KUKA KRL program: EPS_2_25694_BP04_A_20251117072358.src

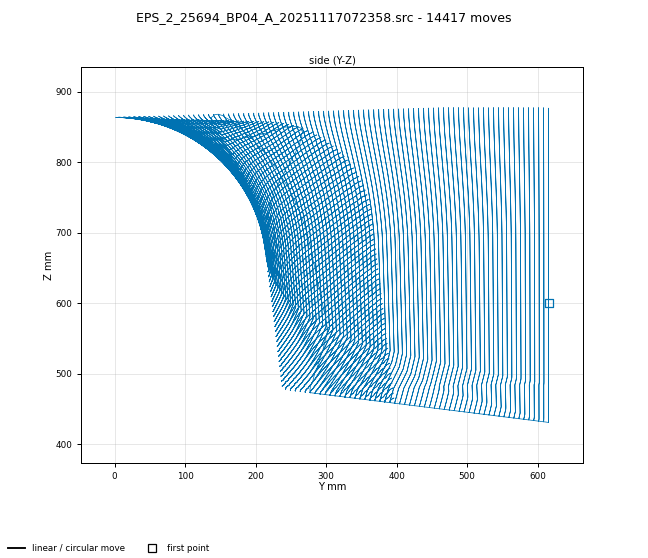
[picture p0: tool path of EPS_2_25694_BP04_A_20251117072358.src, 14417 of 14419 moves have a stored position in this frame; points joined in program order, loops and branches not executed]
&ACCESS RVP
&REL 4
&COMMENT QRS 19112012
&PARAM EDITMASK = *
DEF PART()
EXT BAS (BAS_COMMAND :IN,REAL :IN )
INT I
BAS (#INITMOV,0 )

;KUKA QRS Post kuka4.cps  Date:22-06-2017 !

File_ID=2911

QRS_PRE_INIT()

;Init var - Until changes are made in qrs_pre_init
Outlet_Square_prg=0
Inlet_1_Square_prg=0
Inlet_2_Square_prg=0
Inlet_3_Square_prg=0
Inlet_4_Square_prg=0
Inlet_5_Square_prg=0

Outlet_1={X 0.000, Y 466.000, Z 687.000, B 0.000, E1 0.000 }
Inlet_1={X 0.000, Y 508.730, Z 662.000, B 0.000, E1 180.000 }
Outlet_1_type=381
Inlet_1_type=0
;QRS#1=Sidecore dimensions
;QRS#2=375-15" Concrete
;QRS#3=DeadEnd 381
;QRS#4=
;QRS#5=
;QRS#6=
;QRS#7=
;QRS#8=
;QRS#9=24L PSX-2
;QRS#10=

;QRS#11=
;QRS#12=
;QRS#13=
;QRS#14=
;QRS#15=
;QRS#16=1220x127x1219 4'
;QRS#17=EPS Height
;QRS#18=877,5
;QRS#19=*
;QRS#20= UPDATED VERSION 22-06-2017
;QRS#21=*
Outlet_Square=0150
Inlet_1_Square=00
Inlet_2_Square=0
Inlet_3_Square=0
Inlet_4_Square=0
Inlet_5_Square=0
Mill_Square=1
Outlet_Square_Prg=261
Inlet_1_Square_prg=0

QRS_INIT()

$ADVANCE=5

; T1
PTP {E1 173.596,E2 173.596}
PTP {X 0,Y 615.505,A -85,B 0,C 180,E1 173.596,E2 173.596,E3 0,E4 0,E5 0,E6 0}
QRS_SPEED_INIT()
LIN {X 0,Y 615.505,Z 600,A -85,B 0,C 180,E1 173.596,E2 173.596,E3 0,E4 0,E5 0,E6 0} C_VEL
LIN {X 0,Y 615.505,Z 441.122,A -85,B 0,C 180,E1 173.596,E2 173.596} C_VEL
LIN {X 0,Y 615.505,Z 432.953,A -85,B 0,C 180,E1 173.596,E2 173.596} C_VEL
LIN {X 0,Y 615.487,Z 430.953,A -85,B 0,C 180,E1 173.41,E2 173.41} C_VEL
LIN {X 0,Y 615.475,Z 430.938,A -85,B 0,C 180,E1 170.801,E2 170.801} C_VEL
LIN {X 0,Y 615.486,Z 430.932,A -85,B 0,C 180,E1 168.139,E2 168.139} C_VEL
LIN {X 0,Y 615.48,Z 430.947,A -85,B 0,C 180,E1 165.451,E2 165.451} C_VEL
LIN {X 0,Y 615.476,Z 430.939,A -85,B 0,C 180,E1 162.729,E2 162.729} C_VEL
LIN {X 0,Y 615.485,Z 430.933,A -85,B 0,C 180,E1 159.967,E2 159.967} C_VEL
LIN {X 0,Y 615.486,Z 430.952,A -85,B 0,C 180,E1 157.156,E2 157.156} C_VEL
LIN {X 0,Y 615.484,Z 430.933,A -85,B 0,C 180,E1 154.284,E2 154.284} C_VEL
LIN {X 0,Y 615.476,Z 430.939,A -85,B 0,C 180,E1 151.549,E2 151.549} C_VEL
LIN {X 0,Y 615.483,Z 430.951,A -85,B 0,C 180,E1 148.912,E2 148.912} C_VEL
LIN {X 0,Y 615.496,Z 430.929,A -85,B 0,C 180,E1 145.979,E2 145.979} C_VEL
LIN {X 0,Y 615.487,Z 430.946,A -85,B 0,C 180,E1 143.062,E2 143.062} C_VEL
LIN {X 0,Y 615.474,Z 430.938,A -85,B 0,C 180,E1 140.249,E2 140.249} C_VEL
LIN {X 0,Y 615.488,Z 430.931,A -85,B 0,C 180,E1 137.648,E2 137.648} C_VEL
LIN {X 0,Y 615.48,Z 430.948,A -85,B 0,C 180,E1 134.931,E2 134.931} C_VEL
LIN {X 0,Y 615.477,Z 430.936,A -85,B 0,C 180,E1 132.08,E2 132.08} C_VEL
LIN {X 0,Y 615.493,Z 430.93,A -85,B 0,C 180,E1 129.749,E2 129.749} C_VEL
LIN {X 0,Y 615.478,Z 430.944,A -85,B 0,C 180,E1 126.936,E2 126.936} C_VEL
LIN {X 0,Y 615.49,Z 430.948,A -85,B 0,C 180,E1 124.702,E2 124.702} C_VEL
LIN {X 0,Y 615.484,Z 430.946,A -85,B 0,C 180,E1 122.331,E2 122.331} C_VEL
LIN {X 0,Y 615.493,Z 430.93,A -85,B 0,C 180,E1 119.405,E2 119.405} C_VEL
LIN {X 0,Y 615.491,Z 430.952,A -85,B 0,C 180,E1 116.443,E2 116.443} C_VEL
LIN {X 0,Y 615.487,Z 430.932,A -85,B 0,C 180,E1 113.556,E2 113.556} C_VEL
LIN {X 0,Y 615.477,Z 430.942,A -85,B 0,C 180,E1 110.731,E2 110.731} C_VEL
LIN {X 0,Y 615.478,Z 430.943,A -85,B 0,C 180,E1 107.957,E2 107.957} C_VEL
LIN {X 0,Y 615.488,Z 430.931,A -85,B 0,C 180,E1 105.226,E2 105.226} C_VEL
LIN {X 0,Y 615.479,Z 430.943,A -85,B 0,C 180,E1 102.53,E2 102.53} C_VEL
LIN {X 0,Y 615.48,Z 430.943,A -85,B 0,C 180,E1 99.862,E2 99.862} C_VEL
LIN {X 0,Y 615.489,Z 430.931,A -85,B 0,C 180,E1 97.215,E2 97.215} C_VEL
LIN {X 0,Y 615.476,Z 430.939,A -85,B 0,C 180,E1 94.585,E2 94.585} C_VEL
LIN {X 0,Y 615.493,Z 430.949,A -85,B 0,C 180,E1 91.963,E2 91.963} C_VEL
LIN {X 0,Y 615.474,Z 430.937,A -85,B 0,C 180,E1 89.346,E2 89.346} C_VEL
LIN {X 0,Y 615.484,Z 430.933,A -85,B 0,C 180,E1 86.727,E2 86.727} C_VEL
LIN {X 0,Y 615.484,Z 430.946,A -85,B 0,C 180,E1 84.102,E2 84.102} C_VEL
LIN {X 0,Y 615.477,Z 430.941,A -85,B 0,C 180,E1 81.463,E2 81.463} C_VEL
LIN {X 0,Y 615.497,Z 430.929,A -85,B 0,C 180,E1 78.807,E2 78.807} C_VEL
LIN {X 0,Y 615.48,Z 430.944,A -85,B 0,C 180,E1 76.068,E2 76.068} C_VEL
LIN {X 0,Y 615.477,Z 430.944,A -85,B 0,C 180,E1 73.413,E2 73.413} C_VEL
LIN {X 0,Y 615.485,Z 430.931,A -85,B 0,C 180,E1 70.662,E2 70.662} C_VEL
LIN {X 0,Y 615.478,Z 430.946,A -85,B 0,C 180,E1 67.864,E2 67.864} C_VEL
LIN {X 0,Y 615.475,Z 430.938,A -85,B 0,C 180,E1 65.008,E2 65.008} C_VEL
LIN {X 0,Y 615.481,Z 430.934,A -85,B 0,C 180,E1 62.823,E2 62.823} C_VEL
LIN {X 0,Y 615.476,Z 430.936,A -85,B 0,C 180,E1 60.206,E2 60.206} C_VEL
LIN {X 0,Y 615.489,Z 430.949,A -85,B 0,C 180,E1 57.543,E2 57.543} C_VEL
LIN {X 0,Y 615.483,Z 430.945,A -85,B 0,C 180,E1 55.186,E2 55.186} C_VEL
LIN {X 0,Y 615.474,Z 430.937,A -85,B 0,C 180,E1 52.758,E2 52.758} C_VEL
LIN {X 0,Y 615.476,Z 430.937,A -85,B 0,C 180,E1 49.912,E2 49.912} C_VEL
LIN {X 0,Y 615.478,Z 430.942,A -85,B 0,C 180,E1 47.647,E2 47.647} C_VEL
LIN {X 0,Y 615.48,Z 430.943,A -85,B 0,C 180,E1 44.932,E2 44.932} C_VEL
LIN {X 0,Y 615.49,Z 430.931,A -85,B 0,C 180,E1 42.082,E2 42.082} C_VEL
LIN {X 0,Y 615.493,Z 430.948,A -85,B 0,C 180,E1 39.064,E2 39.064} C_VEL
LIN {X 0,Y 615.479,Z 430.935,A -85,B 0,C 180,E1 36.425,E2 36.425} C_VEL
LIN {X 0,Y 615.476,Z 430.94,A -85,B 0,C 180,E1 33.535,E2 33.535} C_VEL
LIN {X 0,Y 615.485,Z 430.95,A -85,B 0,C 180,E1 30.919,E2 30.919} C_VEL
LIN {X 0,Y 615.476,Z 430.939,A -85,B 0,C 180,E1 28.451,E2 28.451} C_VEL
LIN {X 0,Y 615.484,Z 430.933,A -85,B 0,C 180,E1 25.716,E2 25.716} C_VEL
LIN {X 0,Y 615.486,Z 430.952,A -85,B 0,C 180,E1 22.844,E2 22.844} C_VEL
LIN {X 0,Y 615.485,Z 430.933,A -85,B 0,C 180,E1 20.033,E2 20.033} C_VEL
LIN {X 0,Y 615.476,Z 430.939,A -85,B 0,C 180,E1 17.271,E2 17.271} C_VEL
LIN {X 0,Y 615.484,Z 430.947,A -85,B 0,C 180,E1 14.549,E2 14.549} C_VEL
LIN {X 0,Y 615.486,Z 430.932,A -85,B 0,C 180,E1 11.861,E2 11.861} C_VEL
LIN {X 0,Y 615.475,Z 430.938,A -85,B 0,C 180,E1 9.199,E2 9.199} C_VEL
LIN {X 0,Y 615.489,Z 430.951,A -85,B 0,C 180,E1 6.556,E2 6.556} C_VEL
LIN {X 0,Y 615.477,Z 430.936,A -85,B 0,C 180,E1 3.928,E2 3.928} C_VEL
LIN {X 0,Y 615.484,Z 430.933,A -85,B 0,C 180,E1 1.308,E2 1.308} C_VEL
LIN {X 0,Y 615.483,Z 430.945,A -85,B 0,C 180,E1 -1.309,E2 -1.309} C_VEL
LIN {X 0,Y 615.478,Z 430.942,A -85,B 0,C 180,E1 -3.929,E2 -3.929} C_VEL
LIN {X 0,Y 615.487,Z 430.931,A -85,B 0,C 180,E1 -6.589,E2 -6.589} C_VEL
LIN {X 0,Y 615.474,Z 430.94,A -85,B 0,C 180,E1 -9.199,E2 -9.199} C_VEL
LIN {X 0,Y 615.484,Z 430.948,A -85,B 0,C 180,E1 -11.861,E2 -11.861} C_VEL
LIN {X 0,Y 615.48,Z 430.934,A -85,B 0,C 180,E1 -14.549,E2 -14.549} C_VEL
LIN {X 0,Y 615.475,Z 430.939,A -85,B 0,C 180,E1 -17.271,E2 -17.271} C_VEL
LIN {X 0,Y 615.484,Z 430.946,A -85,B 0,C 180,E1 -20.033,E2 -20.033} C_VEL
LIN {X 0,Y 615.486,Z 430.931,A -85,B 0,C 180,E1 -22.845,E2 -22.845} C_VEL
LIN {X 0,Y 615.483,Z 430.945,A -85,B 0,C 180,E1 -25.716,E2 -25.716} C_VEL
LIN {X 0,Y 615.477,Z 430.94,A -85,B 0,C 180,E1 -28.451,E2 -28.451} C_VEL
LIN {X 0,Y 615.483,Z 430.932,A -85,B 0,C 180,E1 -31.088,E2 -31.088} C_VEL
LIN {X 0,Y 615.495,Z 430.949,A -85,B 0,C 180,E1 -34.021,E2 -34.021} C_VEL
LIN {X 0,Y 615.486,Z 430.932,A -85,B 0,C 180,E1 -36.938,E2 -36.938} C_VEL
LIN {X 0,Y 615.476,Z 430.941,A -85,B 0,C 180,E1 -39.751,E2 -39.751} C_VEL
LIN {X 0,Y 615.489,Z 430.947,A -85,B 0,C 180,E1 -42.353,E2 -42.353} C_VEL
LIN {X 0,Y 615.48,Z 430.934,A -85,B 0,C 180,E1 -45.069,E2 -45.069} C_VEL
LIN {X 0,Y 615.476,Z 430.942,A -85,B 0,C 180,E1 -47.921,E2 -47.921} C_VEL
LIN {X 0,Y 615.491,Z 430.948,A -85,B 0,C 180,E1 -50.251,E2 -50.251} C_VEL
LIN {X 0,Y 615.48,Z 430.935,A -85,B 0,C 180,E1 -53.064,E2 -53.064} C_VEL
LIN {X 0,Y 615.49,Z 430.931,A -85,B 0,C 180,E1 -55.299,E2 -55.299} C_VEL
LIN {X 0,Y 615.484,Z 430.933,A -85,B 0,C 180,E1 -57.669,E2 -57.669} C_VEL
LIN {X 0,Y 615.498,Z 431.074,A -85,B 0,C 180,E1 -60.595,E2 -60.595} C_VEL
LIN {X 0,Y 615.496,Z 431.86,A -85,B 0,C 180,E1 -60.782,E2 -60.782} C_VEL
LIN {X 0,Y 615.493,Z 454.299,A -85,B 0,C 180,E1 -63.557,E2 -63.557} C_VEL
LIN {X 0,Y 615.477,Z 476.35,A -85,B 0,C 180,E1 -66.219,E2 -66.219} C_VEL
LIN {X 0,Y 615.491,Z 484.19,A -85,B 0,C 180,E1 -67.134,E2 -67.134} C_VEL
LIN {X 0,Y 615.489,Z 494.25,A -85,B 0,C 180,E1 -67.28,E2 -67.28} C_VEL
LIN {X 0,Y 615.488,Z 696.741,A -85,B 0,C 180,E1 -69.786,E2 -69.786} C_VEL
LIN {X 0,Y 615.493,Z 712.21,A -85,B 0,C 180,E1 -70.098,E2 -70.098} C_VEL
LIN {X 0,Y 615.492,Z 727.984,A -85,B 0,C 180,E1 -70.533,E2 -70.533} C_VEL
LIN {X 0,Y 615.492,Z 743.625,A -85,B 0,C 180,E1 -71.095,E2 -71.095} C_VEL
LIN {X 0,Y 615.497,Z 759.271,A -85,B 0,C 180,E1 -71.8,E2 -71.8} C_VEL
LIN {X 0,Y 615.499,Z 774.742,A -85,B 0,C 180,E1 -72.645,E2 -72.645} C_VEL
LIN {X 0,Y 615.497,Z 788.923,A -85,B 0,C 180,E1 -73.565,E2 -73.565} C_VEL
LIN {X 0,Y 615.497,Z 802.468,A -85,B 0,C 180,E1 -74.605,E2 -74.605} C_VEL
LIN {X 0,Y 615.496,Z 815.245,A -85,B 0,C 180,E1 -75.759,E2 -75.759} C_VEL
LIN {X 0,Y 615.491,Z 826.671,A -85,B 0,C 180,E1 -76.967,E2 -76.967} C_VEL
LIN {X 0,Y 615.489,Z 837.477,A -85,B 0,C 180,E1 -78.307,E2 -78.307} C_VEL
LIN {X 0,Y 615.49,Z 846.606,A -85,B 0,C 180,E1 -79.64,E2 -79.64} C_VEL
LIN {X 0,Y 615.49,Z 855.145,A -85,B 0,C 180,E1 -81.133,E2 -81.133} C_VEL
LIN {X 0,Y 615.492,Z 862.719,A -85,B 0,C 180,E1 -82.785,E2 -82.785} C_VEL
LIN {X 0,Y 615.487,Z 867.467,A -85,B 0,C 180,E1 -84.102,E2 -84.102} C_VEL
LIN {X 0,Y 615.489,Z 871.26,A -85,B 0,C 180,E1 -85.416,E2 -85.416} C_VEL
LIN {X 0,Y 615.493,Z 873.996,A -85,B 0,C 180,E1 -86.727,E2 -86.727} C_VEL
LIN {X 0,Y 615.494,Z 875.835,A -85,B 0,C 180,E1 -88.037,E2 -88.037} C_VEL
LIN {X 0,Y 615.491,Z 876.738,A -85,B 0,C 180,E1 -89.346,E2 -89.346} C_VEL
LIN {X 0,Y 615.491,Z 876.738,A -85,B 0,C 180,E1 -90.654,E2 -90.654} C_VEL
LIN {X 0,Y 615.494,Z 875.835,A -85,B 0,C 180,E1 -91.963,E2 -91.963} C_VEL
LIN {X 0,Y 615.493,Z 873.996,A -85,B 0,C 180,E1 -93.273,E2 -93.273} C_VEL
LIN {X 0,Y 615.489,Z 871.26,A -85,B 0,C 180,E1 -94.584,E2 -94.584} C_VEL
LIN {X 0,Y 615.491,Z 866.415,A -85,B 0,C 180,E1 -96.227,E2 -96.227} C_VEL
LIN {X 0,Y 615.486,Z 861.303,A -85,B 0,C 180,E1 -97.545,E2 -97.545} C_VEL
LIN {X 0,Y 615.49,Z 855.145,A -85,B 0,C 180,E1 -98.867,E2 -98.867} C_VEL
LIN {X 0,Y 615.489,Z 845.582,A -85,B 0,C 180,E1 -100.527,E2 -100.527} C_VEL
LIN {X 0,Y 615.492,Z 836.244,A -85,B 0,C 180,E1 -101.86,E2 -101.86} C_VEL
LIN {X 0,Y 615.491,Z 826.671,A -85,B 0,C 180,E1 -103.033,E2 -103.033} C_VEL
LIN {X 0,Y 615.496,Z 815.245,A -85,B 0,C 180,E1 -104.241,E2 -104.241} C_VEL
LIN {X 0,Y 615.497,Z 802.468,A -85,B 0,C 180,E1 -105.395,E2 -105.395} C_VEL
LIN {X 0,Y 615.495,Z 788.932,A -85,B 0,C 180,E1 -106.434,E2 -106.434} C_VEL
LIN {X 0,Y 615.498,Z 774.742,A -85,B 0,C 180,E1 -107.355,E2 -107.355} C_VEL
LIN {X 0,Y 615.497,Z 759.271,A -85,B 0,C 180,E1 -108.2,E2 -108.2} C_VEL
LIN {X 0,Y 615.492,Z 743.625,A -85,B 0,C 180,E1 -108.905,E2 -108.905} C_VEL
LIN {X 0,Y 615.492,Z 727.984,A -85,B 0,C 180,E1 -109.467,E2 -109.467} C_VEL
LIN {X 0,Y 615.493,Z 712.21,A -85,B 0,C 180,E1 -109.902,E2 -109.902} C_VEL
LIN {X 0,Y 615.489,Z 695.6,A -85,B 0,C 180,E1 -110.23,E2 -110.23} C_VEL
LIN {X 0,Y 615.49,Z 484.677,A -85,B 0,C 180,E1 -112.844,E2 -112.844} C_VEL
LIN {X 0,Y 615.493,Z 483.482,A -85,B 0,C 180,E1 -112.933,E2 -112.933} C_VEL
LIN {X 0,Y 615.482,Z 460.283,A -85,B 0,C 180,E1 -115.715,E2 -115.715} C_VEL
LIN {X 0,Y 615.495,Z 436.348,A -85,B 0,C 180,E1 -118.657,E2 -118.657} C_VEL
LIN {X 0,Y 615.496,Z 431.31,A -85,B 0,C 180,E1 -119.311,E2 -119.311} C_VEL
LIN {X 0,Y 615.477,Z 430.936,A -85,B 0,C 180,E1 -120.16,E2 -120.16} C_VEL
LIN {X 0,Y 615.489,Z 430.931,A -85,B 0,C 180,E1 -122.457,E2 -122.457} C_VEL
LIN {X 0,Y 615.483,Z 430.933,A -85,B 0,C 180,E1 -124.814,E2 -124.814} C_VEL
LIN {X 0,Y 615.477,Z 430.942,A -85,B 0,C 180,E1 -127.242,E2 -127.242} C_VEL
LIN {X 0,Y 615.476,Z 430.941,A -85,B 0,C 180,E1 -130.088,E2 -130.088} C_VEL
LIN {X 0,Y 615.477,Z 430.936,A -85,B 0,C 180,E1 -132.353,E2 -132.353} C_VEL
LIN {X 0,Y 615.48,Z 430.935,A -85,B 0,C 180,E1 -135.068,E2 -135.068} C_VEL
LIN {X 0,Y 615.489,Z 430.947,A -85,B 0,C 180,E1 -137.918,E2 -137.918} C_VEL
LIN {X 0,Y 615.476,Z 430.941,A -85,B 0,C 180,E1 -140.249,E2 -140.249} C_VEL
LIN {X 0,Y 615.486,Z 430.932,A -85,B 0,C 180,E1 -143.062,E2 -143.062} C_VEL
LIN {X 0,Y 615.495,Z 430.949,A -85,B 0,C 180,E1 -145.979,E2 -145.979} C_VEL
LIN {X 0,Y 615.481,Z 430.933,A -85,B 0,C 180,E1 -148.913,E2 -148.913} C_VEL
LIN {X 0,Y 615.477,Z 430.94,A -85,B 0,C 180,E1 -151.549,E2 -151.549} C_VEL
LIN {X 0,Y 615.483,Z 430.945,A -85,B 0,C 180,E1 -154.284,E2 -154.284} C_VEL
LIN {X 0,Y 615.486,Z 430.931,A -85,B 0,C 180,E1 -157.155,E2 -157.155} C_VEL
LIN {X 0,Y 615.484,Z 430.946,A -85,B 0,C 180,E1 -159.967,E2 -159.967} C_VEL
LIN {X 0,Y 615.475,Z 430.939,A -85,B 0,C 180,E1 -162.729,E2 -162.729} C_VEL
LIN {X 0,Y 615.48,Z 430.934,A -85,B 0,C 180,E1 -165.451,E2 -165.451} C_VEL
LIN {X 0,Y 615.484,Z 430.948,A -85,B 0,C 180,E1 -168.139,E2 -168.139} C_VEL
LIN {X 0,Y 615.474,Z 430.94,A -85,B 0,C 180,E1 -170.801,E2 -170.801} C_VEL
LIN {X 0,Y 615.488,Z 430.931,A -85,B 0,C 180,E1 -173.443,E2 -173.443} C_VEL
LIN {X 0,Y 615.478,Z 430.942,A -85,B 0,C 180,E1 -176.071,E2 -176.071} C_VEL
LIN {X 0,Y 615.483,Z 430.945,A -85,B 0,C 180,E1 -178.691,E2 -178.691} C_VEL
LIN {X 0,Y 615.484,Z 430.933,A -85,B 0,C 180,E1 -181.308,E2 -181.308} C_VEL
LIN {X 0,Y 615.477,Z 430.936,A -85,B 0,C 180,E1 -183.928,E2 -183.928} C_VEL
LIN {X 0,Y 615.487,Z 430.953,A -85,B 0,C 180,E1 -186.59,E2 -186.59} C_VEL
LIN {X 0,Y 614.804,Z 431.086,A -85,B 0,C 180,E1 -187.135,E2 -187.135} C_VEL
LIN {X 0,Y 611.961,Z 431.501,A -85,B 0,C 180,E1 -188.021,E2 -188.021} C_VEL
LIN {X 0,Y 609.57,Z 431.811,A -85,B 0,C 180,E1 -188.734,E2 -188.734} C_VEL
LIN {X 0,Y 608.538,Z 431.928,A -85,B 0,C 180,E1 -189.284,E2 -189.284} C_VEL
LIN {X 0,Y 608.451,Z 431.937,A -85,B 0,C 180,E1 -189.47,E2 -189.47} C_VEL
LIN {X 0,Y 608.46,Z 431.937,A -85,B 0,C 180,E1 -192,E2 -192} C_VEL
LIN {X 0,Y 608.467,Z 431.946,A -85,B 0,C 180,E1 -194.72,E2 -194.72} C_VEL
LIN {X 0,Y 608.445,Z 431.939,A -85,B 0,C 180,E1 -197.477,E2 -197.477} C_VEL
LIN {X 0,Y 608.459,Z 431.938,A -85,B 0,C 180,E1 -200.274,E2 -200.274} C_VEL
LIN {X 0,Y 608.447,Z 431.944,A -85,B 0,C 180,E1 -203.124,E2 -203.124} C_VEL
LIN {X 0,Y 608.465,Z 431.935,A -85,B 0,C 180,E1 -205.722,E2 -205.722} C_VEL
LIN {X 0,Y 608.445,Z 431.938,A -85,B 0,C 180,E1 -208.267,E2 -208.267} C_VEL
LIN {X 0,Y 608.47,Z 431.938,A -85,B 0,C 180,E1 -210.544,E2 -210.544} C_VEL
LIN {X 0,Y 608.45,Z 431.945,A -85,B 0,C 180,E1 -212.88,E2 -212.88} C_VEL
LIN {X 0,Y 608.434,Z 431.947,A -85,B 0,C 180,E1 -215.278,E2 -215.278} C_VEL
LIN {X 0,Y 608.47,Z 431.936,A -85,B 0,C 180,E1 -217.746,E2 -217.746} C_VEL
LIN {X 0,Y 608.473,Z 431.934,A -85,B 0,C 180,E1 -220.333,E2 -220.333} C_VEL
LIN {X 0,Y 608.483,Z 431.943,A -85,B 0,C 180,E1 -223.311,E2 -223.311} C_VEL
LIN {X 0,Y 608.465,Z 431.935,A -85,B 0,C 180,E1 -226.131,E2 -226.131} C_VEL
LIN {X 0,Y 608.447,Z 431.94,A -85,B 0,C 180,E1 -228.824,E2 -228.824} C_VEL
LIN {X 0,Y 608.462,Z 431.946,A -85,B 0,C 180,E1 -231.413,E2 -231.413} C_VEL
LIN {X 0,Y 608.471,Z 431.937,A -85,B 0,C 180,E1 -233.951,E2 -233.951} C_VEL
LIN {X 0,Y 608.466,Z 431.935,A -85,B 0,C 180,E1 -236.33,E2 -236.33} C_VEL
LIN {X 0,Y 608.471,Z 431.935,A -85,B 0,C 180,E1 -238.728,E2 -238.728} C_VEL
LIN {X 0,Y 608.472,Z 431.943,A -85,B 0,C 180,E1 -241.379,E2 -241.379} C_VEL
LIN {X 0,Y 608.467,Z 431.936,A -85,B 0,C 180,E1 -244.279,E2 -244.279} C_VEL
LIN {X 0,Y 608.445,Z 431.938,A -85,B 0,C 180,E1 -246.876,E2 -246.876} C_VEL
LIN {X 0,Y 608.463,Z 431.941,A -85,B 0,C 180,E1 -249.321,E2 -249.321} C_VEL
LIN {X 0,Y 608.442,Z 431.947,A -85,B 0,C 180,E1 -251.828,E2 -251.828} C_VEL
LIN {X 0,Y 608.47,Z 431.935,A -85,B 0,C 180,E1 -254.594,E2 -254.594} C_VEL
LIN {X 0,Y 608.472,Z 431.938,A -85,B 0,C 180,E1 -257.323,E2 -257.323} C_VEL
LIN {X 0,Y 608.449,Z 431.945,A -85,B 0,C 180,E1 -260.023,E2 -260.023} C_VEL
LIN {X 0,Y 608.483,Z 431.933,A -85,B 0,C 180,E1 -262.701,E2 -262.701} C_VEL
LIN {X 0,Y 608.446,Z 431.94,A -85,B 0,C 180,E1 -265.362,E2 -265.362} C_VEL
LIN {X 0,Y 608.463,Z 431.946,A -85,B 0,C 180,E1 -268.014,E2 -268.014} C_VEL
LIN {X 0,Y 608.469,Z 431.936,A -85,B 0,C 180,E1 -270.662,E2 -270.662} C_VEL
LIN {X 0,Y 608.477,Z 431.934,A -85,B 0,C 180,E1 -273.311,E2 -273.311} C_VEL
LIN {X 0,Y 608.457,Z 431.945,A -85,B 0,C 180,E1 -275.967,E2 -275.967} C_VEL
LIN {X 0,Y 608.45,Z 431.94,A -85,B 0,C 180,E1 -278.636,E2 -278.636} C_VEL
LIN {X 0,Y 608.48,Z 431.933,A -85,B 0,C 180,E1 -281.323,E2 -281.323} C_VEL
LIN {X 0,Y 608.464,Z 431.943,A -85,B 0,C 180,E1 -284.037,E2 -284.037} C_VEL
LIN {X 0,Y 608.472,Z 431.937,A -85,B 0,C 180,E1 -286.783,E2 -286.783} C_VEL
LIN {X 0,Y 608.449,Z 431.938,A -85,B 0,C 180,E1 -289.57,E2 -289.57} C_VEL
LIN {X 0,Y 608.454,Z 431.946,A -85,B 0,C 180,E1 -292.476,E2 -292.476} C_VEL
LIN {X 0,Y 608.45,Z 431.945,A -85,B 0,C 180,E1 -294.571,E2 -294.571} C_VEL
LIN {X 0,Y 608.473,Z 431.935,A -85,B 0,C 180,E1 -297.207,E2 -297.207} C_VEL
LIN {X 0,Y 608.457,Z 431.939,A -85,B 0,C 180,E1 -299.971,E2 -299.971} C_VEL
LIN {X 0,Y 608.462,Z 431.947,A -85,B 0,C 180,E1 -302.523,E2 -302.523} C_VEL
LIN {X 0,Y 608.448,Z 431.938,A -85,B 0,C 180,E1 -305.276,E2 -305.276} C_VEL
LIN {X 0,Y 608.46,Z 431.936,A -85,B 0,C 180,E1 -307.746,E2 -307.746} C_VEL
LIN {X 0,Y 608.445,Z 431.943,A -85,B 0,C 180,E1 -310.329,E2 -310.329} C_VEL
LIN {X 0,Y 608.446,Z 431.944,A -85,B 0,C 180,E1 -312.959,E2 -312.959} C_VEL
LIN {X 0,Y 608.459,Z 431.936,A -85,B 0,C 180,E1 -315.735,E2 -315.735} C_VEL
LIN {X 0,Y 608.456,Z 431.945,A -85,B 0,C 180,E1 -318.657,E2 -318.657} C_VEL
LIN {X 0,Y 608.466,Z 431.937,A -85,B 0,C 180,E1 -321.412,E2 -321.412} C_VEL
LIN {X 0,Y 608.469,Z 431.935,A -85,B 0,C 180,E1 -323.95,E2 -323.95} C_VEL
LIN {X 0,Y 608.459,Z 431.937,A -85,B 0,C 180,E1 -326.329,E2 -326.329} C_VEL
LIN {X 0,Y 608.468,Z 431.941,A -85,B 0,C 180,E1 -328.727,E2 -328.727} C_VEL
LIN {X 0,Y 608.465,Z 431.94,A -85,B 0,C 180,E1 -331.379,E2 -331.379} C_VEL
LIN {X 0,Y 608.44,Z 431.938,A -85,B 0,C 180,E1 -333.965,E2 -333.965} C_VEL
LIN {X 0,Y 608.464,Z 431.935,A -85,B 0,C 180,E1 -336.155,E2 -336.155} C_VEL
LIN {X 0,Y 608.453,Z 431.945,A -85,B 0,C 180,E1 -339.019,E2 -339.019} C_VEL
LIN {X 0,Y 608.449,Z 431.939,A -85,B 0,C 180,E1 -341.828,E2 -341.828} C_VEL
LIN {X 0,Y 608.462,Z 431.936,A -85,B 0,C 180,E1 -344.594,E2 -344.594} C_VEL
LIN {X 0,Y 608.472,Z 431.945,A -85,B 0,C 180,E1 -347.323,E2 -347.323} C_VEL
LIN {X 0,Y 608.454,Z 431.938,A -85,B 0,C 180,E1 -350.023,E2 -350.023} C_VEL
LIN {X 0,Y 608.455,Z 431.937,A -85,B 0,C 180,E1 -352.701,E2 -352.701} C_VEL
LIN {X 0,Y 608.465,Z 431.945,A -85,B 0,C 180,E1 -355.363,E2 -355.363} C_VEL
LIN {X 0,Y 608.446,Z 431.94,A -85,B 0,C 180,E1 -358.014,E2 -358.014} C_VEL
LIN {X 0,Y 608.478,Z 431.934,A -85,B 0,C 180,E1 -360.662,E2 -360.662} C_VEL
LIN {X 0,Y 608.472,Z 431.941,A -85,B 0,C 180,E1 -363.311,E2 -363.311} C_VEL
LIN {X 0,Y 608.453,Z 431.941,A -85,B 0,C 180,E1 -365.967,E2 -365.967} C_VEL
LIN {X 0,Y 608.457,Z 431.936,A -85,B 0,C 180,E1 -368.636,E2 -368.636} C_VEL
LIN {X 0,Y 608.467,Z 431.939,A -85,B 0,C 180,E1 -371.324,E2 -371.324} C_VEL
LIN {X 0,Y 608.459,Z 431.942,A -85,B 0,C 180,E1 -374.038,E2 -374.038} C_VEL
LIN {X 0,Y 608.469,Z 431.934,A -85,B 0,C 180,E1 -376.784,E2 -376.784} C_VEL
LIN {X 0,Y 608.444,Z 431.943,A -85,B 0,C 180,E1 -379.571,E2 -379.571} C_VEL
LIN {X 0,Y 608.466,Z 431.938,A -85,B 0,C 180,E1 -382.406,E2 -382.406} C_VEL
LIN {X 0,Y 608.45,Z 431.938,A -85,B 0,C 180,E1 -384.571,E2 -384.571} C_VEL
LIN {X 0,Y 608.474,Z 431.934,A -85,B 0,C 180,E1 -387.209,E2 -387.209} C_VEL
LIN {X 0,Y 608.465,Z 431.945,A -85,B 0,C 180,E1 -389.973,E2 -389.973} C_VEL
LIN {X 0,Y 608.453,Z 431.94,A -85,B 0,C 180,E1 -392.523,E2 -392.523} C_VEL
LIN {X 0,Y 608.433,Z 431.939,A -85,B 0,C 180,E1 -395.278,E2 -395.278} C_VEL
LIN {X 0,Y 608.471,Z 431.939,A -85,B 0,C 180,E1 -397.746,E2 -397.746} C_VEL
LIN {X 0,Y 608.475,Z 431.943,A -85,B 0,C 180,E1 -400.333,E2 -400.333} C_VEL
LIN {X 0,Y 608.483,Z 431.933,A -85,B 0,C 180,E1 -403.312,E2 -403.312} C_VEL
LIN {X 0,Y 608.464,Z 431.944,A -85,B 0,C 180,E1 -406.131,E2 -406.131} C_VEL
LIN {X 0,Y 608.447,Z 431.941,A -85,B 0,C 180,E1 -408.824,E2 -408.824} C_VEL
LIN {X 0,Y 608.462,Z 431.935,A -85,B 0,C 180,E1 -411.413,E2 -411.413} C_VEL
LIN {X 0,Y 608.472,Z 431.938,A -85,B 0,C 180,E1 -413.951,E2 -413.951} C_VEL
LIN {X 0,Y 608.465,Z 431.944,A -85,B 0,C 180,E1 -416.33,E2 -416.33} C_VEL
LIN {X 0,Y 608.472,Z 431.94,A -85,B 0,C 180,E1 -418.728,E2 -418.728} C_VEL
LIN {X 0,Y 608.479,Z 432.113,A -85,B 0,C 180,E1 -420.412,E2 -420.412} C_VEL
LIN {X 0,Y 608.762,Z 434.852,A -85,B 0,C 180,E1 -420.807,E2 -420.807} C_VEL
LIN {X 0,Y 608.713,Z 457.291,A -85,B 0,C 180,E1 -423.609,E2 -423.609} C_VEL
LIN {X 0,Y 608.652,Z 479.731,A -85,B 0,C 180,E1 -426.344,E2 -426.344} C_VEL
LIN {X 0,Y 608.707,Z 484.388,A -85,B 0,C 180,E1 -426.876,E2 -426.876} C_VEL
LIN {X 0,Y 608.966,Z 488.161,A -85,B 0,C 180,E1 -426.947,E2 -426.947} C_VEL
LIN {X 0,Y 608.839,Z 696.739,A -85,B 0,C 180,E1 -429.556,E2 -429.556} C_VEL
LIN {X 0,Y 608.806,Z 713.133,A -85,B 0,C 180,E1 -429.892,E2 -429.892} C_VEL
LIN {X 0,Y 608.775,Z 730.575,A -85,B 0,C 180,E1 -430.397,E2 -430.397} C_VEL
LIN {X 0,Y 608.717,Z 745.782,A -85,B 0,C 180,E1 -430.964,E2 -430.964} C_VEL
LIN {X 0,Y 608.691,Z 760.918,A -85,B 0,C 180,E1 -431.672,E2 -431.672} C_VEL
LIN {X 0,Y 608.646,Z 776.158,A -85,B 0,C 180,E1 -432.53,E2 -432.53} C_VEL
LIN {X 0,Y 608.583,Z 789.741,A -85,B 0,C 180,E1 -433.434,E2 -433.434} C_VEL
LIN {X 0,Y 608.565,Z 802.486,A -85,B 0,C 180,E1 -434.425,E2 -434.425} C_VEL
LIN {X 0,Y 608.523,Z 813.841,A -85,B 0,C 180,E1 -435.452,E2 -435.452} C_VEL
LIN {X 0,Y 608.489,Z 825.297,A -85,B 0,C 180,E1 -436.644,E2 -436.644} C_VEL
LIN {X 0,Y 608.477,Z 835.173,A -85,B 0,C 180,E1 -437.832,E2 -437.832} C_VEL
LIN {X 0,Y 608.454,Z 844.797,A -85,B 0,C 180,E1 -439.195,E2 -439.195} C_VEL
LIN {X 0,Y 608.458,Z 851.852,A -85,B 0,C 180,E1 -440.359,E2 -440.359} C_VEL
LIN {X 0,Y 608.448,Z 858.742,A -85,B 0,C 180,E1 -441.699,E2 -441.699} C_VEL
LIN {X 0,Y 608.436,Z 864.429,A -85,B 0,C 180,E1 -443.034,E2 -443.034} C_VEL
LIN {X 0,Y 608.427,Z 869.017,A -85,B 0,C 180,E1 -444.366,E2 -444.366} C_VEL
LIN {X 0,Y 608.422,Z 871.79,A -85,B 0,C 180,E1 -445.362,E2 -445.362} C_VEL
LIN {X 0,Y 608.42,Z 874.571,A -85,B 0,C 180,E1 -446.689,E2 -446.689} C_VEL
LIN {X 0,Y 608.438,Z 876.433,A -85,B 0,C 180,E1 -448.014,E2 -448.014} C_VEL
LIN {X 0,Y 608.434,Z 877.35,A -85,B 0,C 180,E1 -449.338,E2 -449.338} C_VEL
LIN {X 0,Y 608.434,Z 877.35,A -85,B 0,C 180,E1 -450.662,E2 -450.662} C_VEL
LIN {X 0,Y 608.438,Z 876.433,A -85,B 0,C 180,E1 -451.986,E2 -451.986} C_VEL
LIN {X 0,Y 608.421,Z 874.571,A -85,B 0,C 180,E1 -453.311,E2 -453.311} C_VEL
LIN {X 0,Y 608.422,Z 871.79,A -85,B 0,C 180,E1 -454.638,E2 -454.638} C_VEL
LIN {X 0,Y 608.427,Z 867.956,A -85,B 0,C 180,E1 -455.967,E2 -455.967} C_VEL
LIN {X 0,Y 608.454,Z 863.142,A -85,B 0,C 180,E1 -457.299,E2 -457.299} C_VEL
LIN {X 0,Y 608.446,Z 857.124,A -85,B 0,C 180,E1 -458.636,E2 -458.636} C_VEL
LIN {X 0,Y 608.461,Z 848.901,A -85,B 0,C 180,E1 -460.145,E2 -460.145} C_VEL
LIN {X 0,Y 608.466,Z 840.145,A -85,B 0,C 180,E1 -461.492,E2 -461.492} C_VEL
LIN {X 0,Y 608.496,Z 829.73,A -85,B 0,C 180,E1 -462.846,E2 -462.846} C_VEL
LIN {X 0,Y 608.517,Z 818.978,A -85,B 0,C 180,E1 -464.036,E2 -464.036} C_VEL
LIN {X 0,Y 608.551,Z 806.422,A -85,B 0,C 180,E1 -465.232,E2 -465.232} C_VEL
LIN {X 0,Y 608.578,Z 792.543,A -85,B 0,C 180,E1 -466.358,E2 -466.358} C_VEL
LIN {X 0,Y 608.635,Z 778.979,A -85,B 0,C 180,E1 -467.297,E2 -467.297} C_VEL
LIN {X 0,Y 608.677,Z 764.116,A -85,B 0,C 180,E1 -468.164,E2 -468.164} C_VEL
LIN {X 0,Y 608.709,Z 749.732,A -85,B 0,C 180,E1 -468.861,E2 -468.861} C_VEL
LIN {X 0,Y 608.772,Z 734.453,A -85,B 0,C 180,E1 -469.472,E2 -469.472} C_VEL
LIN {X 0,Y 608.789,Z 718.343,A -85,B 0,C 180,E1 -469.976,E2 -469.976} C_VEL
LIN {X 0,Y 608.815,Z 702.228,A -85,B 0,C 180,E1 -470.345,E2 -470.345} C_VEL
LIN {X 0,Y 608.849,Z 682.029,A -85,B 0,C 180,E1 -470.644,E2 -470.644} C_VEL
LIN {X 0,Y 608.961,Z 486.016,A -85,B 0,C 180,E1 -473.08,E2 -473.08} C_VEL
LIN {X 0,Y 608.653,Z 483.899,A -85,B 0,C 180,E1 -473.16,E2 -473.16} C_VEL
LIN {X 0,Y 608.683,Z 461.863,A -85,B 0,C 180,E1 -475.83,E2 -475.83} C_VEL
LIN {X 0,Y 608.755,Z 438.198,A -85,B 0,C 180,E1 -478.771,E2 -478.771} C_VEL
LIN {X 0,Y 608.559,Z 432.448,A -85,B 0,C 180,E1 -479.512,E2 -479.512} C_VEL
LIN {X 0,Y 608.472,Z 431.986,A -85,B 0,C 180,E1 -479.683,E2 -479.683} C_VEL
LIN {X 0,Y 608.462,Z 431.936,A -85,B 0,C 180,E1 -482.523,E2 -482.523} C_VEL
LIN {X 0,Y 608.447,Z 431.943,A -85,B 0,C 180,E1 -485.276,E2 -485.276} C_VEL
LIN {X 0,Y 608.461,Z 431.944,A -85,B 0,C 180,E1 -487.746,E2 -487.746} C_VEL
LIN {X 0,Y 608.445,Z 431.939,A -85,B 0,C 180,E1 -490.328,E2 -490.328} C_VEL
LIN {X 0,Y 608.465,Z 431.939,A -85,B 0,C 180,E1 -493.309,E2 -493.309} C_VEL
LIN {X 0,Y 608.468,Z 431.939,A -85,B 0,C 180,E1 -496.131,E2 -496.131} C_VEL
LIN {X 0,Y 608.453,Z 431.936,A -85,B 0,C 180,E1 -498.823,E2 -498.823} C_VEL
LIN {X 0,Y 608.467,Z 431.939,A -85,B 0,C 180,E1 -501.412,E2 -501.412} C_VEL
LIN {X 0,Y 608.47,Z 431.944,A -85,B 0,C 180,E1 -503.95,E2 -503.95} C_VEL
LIN {X 0,Y 608.459,Z 431.94,A -85,B 0,C 180,E1 -506.329,E2 -506.329} C_VEL
LIN {X 0,Y 608.469,Z 431.935,A -85,B 0,C 180,E1 -508.727,E2 -508.727} C_VEL
LIN {X 0,Y 608.465,Z 431.936,A -85,B 0,C 180,E1 -511.379,E2 -511.379} C_VEL
LIN {X 0,Y 608.44,Z 431.948,A -85,B 0,C 180,E1 -513.964,E2 -513.964} C_VEL
LIN {X 0,Y 608.464,Z 431.945,A -85,B 0,C 180,E1 -516.155,E2 -516.155} C_VEL
LIN {X 0,Y 608.453,Z 431.936,A -85,B 0,C 180,E1 -519.018,E2 -519.018} C_VEL
LIN {X 0,Y 608.449,Z 431.941,A -85,B 0,C 180,E1 -521.828,E2 -521.828} C_VEL
LIN {X 0,Y 608.462,Z 431.94,A -85,B 0,C 180,E1 -524.594,E2 -524.594} C_VEL
LIN {X 0,Y 608.472,Z 431.934,A -85,B 0,C 180,E1 -527.323,E2 -527.323} C_VEL
LIN {X 0,Y 608.455,Z 431.942,A -85,B 0,C 180,E1 -530.023,E2 -530.023} C_VEL
LIN {X 0,Y 608.455,Z 431.942,A -85,B 0,C 180,E1 -532.7,E2 -532.7} C_VEL
LIN {X 0,Y 608.467,Z 431.935,A -85,B 0,C 180,E1 -535.362,E2 -535.362} C_VEL
LIN {X 0,Y 608.447,Z 431.941,A -85,B 0,C 180,E1 -538.014,E2 -538.014} C_VEL
LIN {X 0,Y 608.478,Z 431.941,A -85,B 0,C 180,E1 -540.662,E2 -540.662} C_VEL
LIN {X 0,Y 608.473,Z 431.935,A -85,B 0,C 180,E1 -543.311,E2 -543.311} C_VEL
LIN {X 0,Y 608.476,Z 431.935,A -85,B 0,C 180,E1 -545.967,E2 -545.967} C_VEL
LIN {X 0,Y 608.458,Z 431.948,A -85,B 0,C 180,E1 -548.636,E2 -548.636} C_VEL
LIN {X 0,Y 608.451,Z 431.937,A -85,B 0,C 180,E1 -549.47,E2 -549.47} C_VEL
LIN {X 0,Y 607.777,Z 432.023,A -85,B 0,C 180,E1 -550.023,E2 -550.023} C_VEL
LIN {X 0,Y 604.925,Z 432.382,A -85,B 0,C 180,E1 -550.92,E2 -550.92} C_VEL
LIN {X 0,Y 602.521,Z 432.679,A -85,B 0,C 180,E1 -551.641,E2 -551.641} C_VEL
LIN {X 0,Y 601.49,Z 432.806,A -85,B 0,C 180,E1 -552.198,E2 -552.198} C_VEL
LIN {X 0,Y 601.406,Z 432.818,A -85,B 0,C 180,E1 -552.386,E2 -552.386} C_VEL
LIN {X 0,Y 601.422,Z 432.82,A -85,B 0,C 180,E1 -554.897,E2 -554.897} C_VEL
LIN {X 0,Y 601.425,Z 432.82,A -85,B 0,C 180,E1 -556.986,E2 -556.986} C_VEL
LIN {X 0,Y 601.4,Z 432.815,A -85,B 0,C 180,E1 -559.809,E2 -559.809} C_VEL
LIN {X 0,Y 601.404,Z 432.821,A -85,B 0,C 180,E1 -562.606,E2 -562.606} C_VEL
LIN {X 0,Y 601.398,Z 432.826,A -85,B 0,C 180,E1 -564.878,E2 -564.878} C_VEL
LIN {X 0,Y 601.415,Z 432.812,A -85,B 0,C 180,E1 -567.867,E2 -567.867} C_VEL
LIN {X 0,Y 601.439,Z 432.811,A -85,B 0,C 180,E1 -570.163,E2 -570.163} C_VEL
LIN {X 0,Y 601.414,Z 432.819,A -85,B 0,C 180,E1 -572.716,E2 -572.716} C_VEL
LIN {X 0,Y 601.402,Z 432.826,A -85,B 0,C 180,E1 -575.115,E2 -575.115} C_VEL
LIN {X 0,Y 601.429,Z 432.817,A -85,B 0,C 180,E1 -577.419,E2 -577.419} C_VEL
LIN {X 0,Y 601.407,Z 432.815,A -85,B 0,C 180,E1 -579.995,E2 -579.995} C_VEL
LIN {X 0,Y 601.408,Z 432.817,A -85,B 0,C 180,E1 -582.67,E2 -582.67} C_VEL
LIN {X 0,Y 601.417,Z 432.82,A -85,B 0,C 180,E1 -585.482,E2 -585.482} C_VEL
LIN {X 0,Y 601.417,Z 432.813,A -85,B 0,C 180,E1 -588.407,E2 -588.407} C_VEL
LIN {X 0,Y 601.428,Z 432.815,A -85,B 0,C 180,E1 -590.876,E2 -590.876} C_VEL
LIN {X 0,Y 601.437,Z 432.816,A -85,B 0,C 180,E1 -593.734,E2 -593.734} C_VEL
LIN {X 0,Y 601.426,Z 432.813,A -85,B 0,C 180,E1 -596.687,E2 -596.687} C_VEL
LIN {X 0,Y 601.423,Z 432.816,A -85,B 0,C 180,E1 -599.059,E2 -599.059} C_VEL
LIN {X 0,Y 601.431,Z 432.82,A -85,B 0,C 180,E1 -601.374,E2 -601.374} C_VEL
LIN {X 0,Y 601.409,Z 432.816,A -85,B 0,C 180,E1 -604.132,E2 -604.132} C_VEL
LIN {X 0,Y 601.415,Z 432.814,A -85,B 0,C 180,E1 -606.59,E2 -606.59} C_VEL
LIN {X 0,Y 601.427,Z 432.82,A -85,B 0,C 180,E1 -609.479,E2 -609.479} C_VEL
LIN {X 0,Y 601.397,Z 432.817,A -85,B 0,C 180,E1 -612.312,E2 -612.312} C_VEL
LIN {X 0,Y 601.413,Z 432.815,A -85,B 0,C 180,E1 -614.409,E2 -614.409} C_VEL
LIN {X 0,Y 601.419,Z 432.815,A -85,B 0,C 180,E1 -617.172,E2 -617.172} C_VEL
LIN {X 0,Y 601.427,Z 432.822,A -85,B 0,C 180,E1 -619.905,E2 -619.905} C_VEL
LIN {X 0,Y 601.452,Z 432.81,A -85,B 0,C 180,E1 -622.615,E2 -622.615} C_VEL
LIN {X 0,Y 601.415,Z 432.815,A -85,B 0,C 180,E1 -625.308,E2 -625.308} C_VEL
LIN {X 0,Y 601.431,Z 432.823,A -85,B 0,C 180,E1 -627.991,E2 -627.991} C_VEL
LIN {X 0,Y 601.441,Z 432.812,A -85,B 0,C 180,E1 -630.67,E2 -630.67} C_VEL
LIN {X 0,Y 601.429,Z 432.813,A -85,B 0,C 180,E1 -633.349,E2 -633.349} C_VEL
LIN {X 0,Y 601.408,Z 432.825,A -85,B 0,C 180,E1 -636.037,E2 -636.037} C_VEL
LIN {X 0,Y 601.435,Z 432.821,A -85,B 0,C 180,E1 -638.061,E2 -638.061} C_VEL
LIN {X 0,Y 601.421,Z 432.813,A -85,B 0,C 180,E1 -641.012,E2 -641.012} C_VEL
LIN {X 0,Y 601.421,Z 432.814,A -85,B 0,C 180,E1 -643.515,E2 -643.515} C_VEL
LIN {X 0,Y 601.435,Z 432.822,A -85,B 0,C 180,E1 -646.287,E2 -646.287} C_VEL
LIN {X 0,Y 601.413,Z 432.814,A -85,B 0,C 180,E1 -649.099,E2 -649.099} C_VEL
LIN {X 0,Y 601.405,Z 432.815,A -85,B 0,C 180,E1 -651.239,E2 -651.239} C_VEL
LIN {X 0,Y 601.451,Z 432.815,A -85,B 0,C 180,E1 -654.14,E2 -654.14} C_VEL
LIN {X 0,Y 601.446,Z 432.811,A -85,B 0,C 180,E1 -657.111,E2 -657.111} C_VEL
LIN {X 0,Y 601.416,Z 432.814,A -85,B 0,C 180,E1 -659.393,E2 -659.393} C_VEL
LIN {X 0,Y 601.409,Z 432.815,A -85,B 0,C 180,E1 -661.726,E2 -661.726} C_VEL
LIN {X 0,Y 601.428,Z 432.815,A -85,B 0,C 180,E1 -664.118,E2 -664.118} C_VEL
LIN {X 0,Y 601.406,Z 432.826,A -85,B 0,C 180,E1 -666.582,E2 -666.582} C_VEL
LIN {X 0,Y 601.435,Z 432.811,A -85,B 0,C 180,E1 -669.536,E2 -669.536} C_VEL
LIN {X 0,Y 601.404,Z 432.824,A -85,B 0,C 180,E1 -672.591,E2 -672.591} C_VEL
LIN {X 0,Y 601.415,Z 432.821,A -85,B 0,C 180,E1 -674.535,E2 -674.535} C_VEL
LIN {X 0,Y 601.408,Z 432.817,A -85,B 0,C 180,E1 -677.33,E2 -677.33} C_VEL
LIN {X 0,Y 601.407,Z 432.815,A -85,B 0,C 180,E1 -680.005,E2 -680.005} C_VEL
LIN {X 0,Y 601.43,Z 432.818,A -85,B 0,C 180,E1 -682.617,E2 -682.617} C_VEL
LIN {X 0,Y 601.428,Z 432.818,A -85,B 0,C 180,E1 -685.069,E2 -685.069} C_VEL
LIN {X 0,Y 601.421,Z 432.815,A -85,B 0,C 180,E1 -687.484,E2 -687.484} C_VEL
LIN {X 0,Y 601.439,Z 432.811,A -85,B 0,C 180,E1 -689.848,E2 -689.848} C_VEL
LIN {X 0,Y 601.446,Z 432.817,A -85,B 0,C 180,E1 -692.889,E2 -692.889} C_VEL
LIN {X 0,Y 601.453,Z 432.809,A -85,B 0,C 180,E1 -695.86,E2 -695.86} C_VEL
LIN {X 0,Y 601.402,Z 432.819,A -85,B 0,C 180,E1 -698.761,E2 -698.761} C_VEL
LIN {X 0,Y 601.418,Z 432.817,A -85,B 0,C 180,E1 -701.608,E2 -701.608} C_VEL
LIN {X 0,Y 601.407,Z 432.814,A -85,B 0,C 180,E1 -704.409,E2 -704.409} C_VEL
LIN {X 0,Y 601.417,Z 432.822,A -85,B 0,C 180,E1 -707.172,E2 -707.172} C_VEL
LIN {X 0,Y 601.431,Z 432.813,A -85,B 0,C 180,E1 -709.905,E2 -709.905} C_VEL
LIN {X 0,Y 601.432,Z 432.812,A -85,B 0,C 180,E1 -712.615,E2 -712.615} C_VEL
LIN {X 0,Y 601.43,Z 432.82,A -85,B 0,C 180,E1 -715.308,E2 -715.308} C_VEL
LIN {X 0,Y 601.416,Z 432.815,A -85,B 0,C 180,E1 -717.991,E2 -717.991} C_VEL
LIN {X 0,Y 601.448,Z 432.809,A -85,B 0,C 180,E1 -720.67,E2 -720.67} C_VEL
LIN {X 0,Y 601.424,Z 432.819,A -85,B 0,C 180,E1 -723.35,E2 -723.35} C_VEL
LIN {X 0,Y 601.406,Z 432.818,A -85,B 0,C 180,E1 -726.037,E2 -726.037} C_VEL
LIN {X 0,Y 601.435,Z 432.81,A -85,B 0,C 180,E1 -728.738,E2 -728.738} C_VEL
LIN {X 0,Y 601.426,Z 432.819,A -85,B 0,C 180,E1 -731.458,E2 -731.458} C_VEL
LIN {X 0,Y 601.409,Z 432.817,A -85,B 0,C 180,E1 -734.206,E2 -734.206} C_VEL
LIN {X 0,Y 601.425,Z 432.812,A -85,B 0,C 180,E1 -736.986,E2 -736.986} C_VEL
LIN {X 0,Y 601.4,Z 432.824,A -85,B 0,C 180,E1 -739.81,E2 -739.81} C_VEL
LIN {X 0,Y 601.405,Z 432.815,A -85,B 0,C 180,E1 -742.606,E2 -742.606} C_VEL
LIN {X 0,Y 601.398,Z 432.815,A -85,B 0,C 180,E1 -744.879,E2 -744.879} C_VEL
LIN {X 0,Y 601.415,Z 432.822,A -85,B 0,C 180,E1 -747.868,E2 -747.868} C_VEL
LIN {X 0,Y 601.44,Z 432.819,A -85,B 0,C 180,E1 -750.163,E2 -750.163} C_VEL
LIN {X 0,Y 601.414,Z 432.815,A -85,B 0,C 180,E1 -752.716,E2 -752.716} C_VEL
LIN {X 0,Y 601.402,Z 432.814,A -85,B 0,C 180,E1 -755.115,E2 -755.115} C_VEL
LIN {X 0,Y 601.431,Z 432.812,A -85,B 0,C 180,E1 -757.419,E2 -757.419} C_VEL
LIN {X 0,Y 601.408,Z 432.822,A -85,B 0,C 180,E1 -759.995,E2 -759.995} C_VEL
LIN {X 0,Y 601.409,Z 432.818,A -85,B 0,C 180,E1 -762.67,E2 -762.67} C_VEL
LIN {X 0,Y 601.419,Z 432.813,A -85,B 0,C 180,E1 -765.483,E2 -765.483} C_VEL
LIN {X 0,Y 601.417,Z 432.823,A -85,B 0,C 180,E1 -768.407,E2 -768.407} C_VEL
LIN {X 0,Y 601.429,Z 432.813,A -85,B 0,C 180,E1 -770.876,E2 -770.876} C_VEL
LIN {X 0,Y 601.438,Z 432.812,A -85,B 0,C 180,E1 -773.734,E2 -773.734} C_VEL
LIN {X 0,Y 601.426,Z 432.82,A -85,B 0,C 180,E1 -776.687,E2 -776.687} C_VEL
LIN {X 0,Y 601.424,Z 432.811,A -85,B 0,C 180,E1 -779.059,E2 -779.059} C_VEL
LIN {X 0,Y 601.454,Z 432.951,A -85,B 0,C 180,E1 -780.132,E2 -780.132} C_VEL
LIN {X 0,Y 602.041,Z 436.348,A -85,B 0,C 180,E1 -780.641,E2 -780.641} C_VEL
LIN {X 0,Y 601.93,Z 458.787,A -85,B 0,C 180,E1 -783.475,E2 -783.475} C_VEL
LIN {X 0,Y 601.824,Z 481.227,A -85,B 0,C 180,E1 -786.242,E2 -786.242} C_VEL
LIN {X 0,Y 601.856,Z 484.396,A -85,B 0,C 180,E1 -786.597,E2 -786.597} C_VEL
LIN {X 0,Y 602.445,Z 487.807,A -85,B 0,C 180,E1 -786.678,E2 -786.678} C_VEL
LIN {X 0,Y 602.179,Z 696.903,A -85,B 0,C 180,E1 -789.323,E2 -789.323} C_VEL
LIN {X 0,Y 602.14,Z 713.143,A -85,B 0,C 180,E1 -789.66,E2 -789.66} C_VEL
LIN {X 0,Y 602.058,Z 730.58,A -85,B 0,C 180,E1 -790.169,E2 -790.169} C_VEL
LIN {X 0,Y 601.976,Z 745.769,A -85,B 0,C 180,E1 -790.743,E2 -790.743} C_VEL
LIN {X 0,Y 601.908,Z 760.819,A -85,B 0,C 180,E1 -791.453,E2 -791.453} C_VEL
LIN {X 0,Y 601.781,Z 776.163,A -85,B 0,C 180,E1 -792.324,E2 -792.324} C_VEL
LIN {X 0,Y 601.697,Z 790.443,A -85,B 0,C 180,E1 -793.292,E2 -793.292} C_VEL
LIN {X 0,Y 601.616,Z 802.49,A -85,B 0,C 180,E1 -794.241,E2 -794.241} C_VEL
LIN {X 0,Y 601.558,Z 813.839,A -85,B 0,C 180,E1 -795.28,E2 -795.28} C_VEL
LIN {X 0,Y 601.488,Z 825.3,A -85,B 0,C 180,E1 -796.486,E2 -796.486} C_VEL
LIN {X 0,Y 601.435,Z 836.429,A -85,B 0,C 180,E1 -797.858,E2 -797.858} C_VEL
LIN {X 0,Y 601.402,Z 845.831,A -85,B 0,C 180,E1 -799.224,E2 -799.224} C_VEL
LIN {X 0,Y 601.364,Z 853.669,A -85,B 0,C 180,E1 -800.583,E2 -800.583} C_VEL
LIN {X 0,Y 601.36,Z 860.294,A -85,B 0,C 180,E1 -801.938,E2 -801.938} C_VEL
LIN {X 0,Y 601.349,Z 866.12,A -85,B 0,C 180,E1 -803.411,E2 -803.411} C_VEL
LIN {X 0,Y 601.347,Z 870.016,A -85,B 0,C 180,E1 -804.635,E2 -804.635} C_VEL
LIN {X 0,Y 601.338,Z 873.288,A -85,B 0,C 180,E1 -805.979,E2 -805.979} C_VEL
LIN {X 0,Y 601.316,Z 875.652,A -85,B 0,C 180,E1 -807.32,E2 -807.32} C_VEL
LIN {X 0,Y 601.34,Z 876.994,A -85,B 0,C 180,E1 -808.661,E2 -808.661} C_VEL
LIN {X 0,Y 601.33,Z 877.5,A -85,B 0,C 180,E1 -810,E2 -810} C_VEL
LIN {X 0,Y 601.34,Z 876.994,A -85,B 0,C 180,E1 -811.339,E2 -811.339} C_VEL
LIN {X 0,Y 601.316,Z 875.652,A -85,B 0,C 180,E1 -812.68,E2 -812.68} C_VEL
LIN {X 0,Y 601.337,Z 873.288,A -85,B 0,C 180,E1 -814.021,E2 -814.021} C_VEL
LIN {X 0,Y 601.347,Z 870.016,A -85,B 0,C 180,E1 -815.365,E2 -815.365} C_VEL
LIN {X 0,Y 601.365,Z 864.429,A -85,B 0,C 180,E1 -817.048,E2 -817.048} C_VEL
LIN {X 0,Y 601.363,Z 858.745,A -85,B 0,C 180,E1 -818.4,E2 -818.4} C_VEL
LIN {X 0,Y 601.4,Z 851.851,A -85,B 0,C 180,E1 -819.755,E2 -819.755} C_VEL
LIN {X 0,Y 601.4,Z 843.485,A -85,B 0,C 180,E1 -821.133,E2 -821.133} C_VEL
LIN {X 0,Y 601.463,Z 833.813,A -85,B 0,C 180,E1 -822.484,E2 -822.484} C_VEL
LIN {X 0,Y 601.521,Z 822.904,A -85,B 0,C 180,E1 -823.786,E2 -823.786} C_VEL
LIN {X 0,Y 601.594,Z 810.283,A -85,B 0,C 180,E1 -825.066,E2 -825.066} C_VEL
LIN {X 0,Y 601.66,Z 796.122,A -85,B 0,C 180,E1 -826.28,E2 -826.28} C_VEL
LIN {X 0,Y 601.756,Z 781.632,A -85,B 0,C 180,E1 -827.326,E2 -827.326} C_VEL
LIN {X 0,Y 601.849,Z 767.252,A -85,B 0,C 180,E1 -828.202,E2 -828.202} C_VEL
LIN {X 0,Y 601.936,Z 751.487,A -85,B 0,C 180,E1 -829.003,E2 -829.003} C_VEL
LIN {X 0,Y 602.046,Z 735.7,A -85,B 0,C 180,E1 -829.654,E2 -829.654} C_VEL
LIN {X 0,Y 602.114,Z 719.854,A -85,B 0,C 180,E1 -830.163,E2 -830.163} C_VEL
LIN {X 0,Y 602.162,Z 703.446,A -85,B 0,C 180,E1 -830.556,E2 -830.556} C_VEL
LIN {X 0,Y 602.21,Z 685.909,A -85,B 0,C 180,E1 -830.834,E2 -830.834} C_VEL
LIN {X 0,Y 602.42,Z 487.807,A -85,B 0,C 180,E1 -833.323,E2 -833.323} C_VEL
LIN {X 0,Y 601.822,Z 484.204,A -85,B 0,C 180,E1 -833.416,E2 -833.416} C_VEL
LIN {X 0,Y 601.879,Z 463.347,A -85,B 0,C 180,E1 -835.959,E2 -835.959} C_VEL
LIN {X 0,Y 602.041,Z 438.707,A -85,B 0,C 180,E1 -839.057,E2 -839.057} C_VEL
LIN {X 0,Y 601.892,Z 434.852,A -85,B 0,C 180,E1 -839.559,E2 -839.559} C_VEL
LIN {X 0,Y 601.453,Z 432.936,A -85,B 0,C 180,E1 -839.868,E2 -839.868} C_VEL
LIN {X 0,Y 601.422,Z 432.815,A -85,B 0,C 180,E1 -842.716,E2 -842.716} C_VEL
LIN {X 0,Y 601.411,Z 432.817,A -85,B 0,C 180,E1 -845.114,E2 -845.114} C_VEL
LIN {X 0,Y 601.429,Z 432.82,A -85,B 0,C 180,E1 -847.418,E2 -847.418} C_VEL
LIN {X 0,Y 601.405,Z 432.82,A -85,B 0,C 180,E1 -849.994,E2 -849.994} C_VEL
LIN {X 0,Y 601.405,Z 432.814,A -85,B 0,C 180,E1 -852.67,E2 -852.67} C_VEL
LIN {X 0,Y 601.419,Z 432.819,A -85,B 0,C 180,E1 -855.482,E2 -855.482} C_VEL
LIN {X 0,Y 601.421,Z 432.814,A -85,B 0,C 180,E1 -858.406,E2 -858.406} C_VEL
LIN {X 0,Y 601.433,Z 432.811,A -85,B 0,C 180,E1 -860.875,E2 -860.875} C_VEL
LIN {X 0,Y 601.437,Z 432.819,A -85,B 0,C 180,E1 -863.733,E2 -863.733} C_VEL
LIN {X 0,Y 601.42,Z 432.813,A -85,B 0,C 180,E1 -866.686,E2 -866.686} C_VEL
LIN {X 0,Y 601.425,Z 432.812,A -85,B 0,C 180,E1 -869.058,E2 -869.058} C_VEL
LIN {X 0,Y 601.425,Z 432.812,A -85,B 0,C 180,E1 -871.373,E2 -871.373} C_VEL
LIN {X 0,Y 601.398,Z 432.819,A -85,B 0,C 180,E1 -873.636,E2 -873.636} C_VEL
LIN {X 0,Y 601.416,Z 432.816,A -85,B 0,C 180,E1 -876.59,E2 -876.59} C_VEL
LIN {X 0,Y 601.426,Z 432.811,A -85,B 0,C 180,E1 -879.478,E2 -879.478} C_VEL
LIN {X 0,Y 601.393,Z 432.825,A -85,B 0,C 180,E1 -882.312,E2 -882.312} C_VEL
LIN {X 0,Y 601.407,Z 432.822,A -85,B 0,C 180,E1 -884.409,E2 -884.409} C_VEL
LIN {X 0,Y 601.416,Z 432.813,A -85,B 0,C 180,E1 -887.172,E2 -887.172} C_VEL
LIN {X 0,Y 601.432,Z 432.815,A -85,B 0,C 180,E1 -889.905,E2 -889.905} C_VEL
LIN {X 0,Y 601.432,Z 432.818,A -85,B 0,C 180,E1 -892.615,E2 -892.615} C_VEL
LIN {X 0,Y 601.432,Z 432.811,A -85,B 0,C 180,E1 -895.308,E2 -895.308} C_VEL
LIN {X 0,Y 601.417,Z 432.816,A -85,B 0,C 180,E1 -897.991,E2 -897.991} C_VEL
LIN {X 0,Y 601.448,Z 432.816,A -85,B 0,C 180,E1 -900.669,E2 -900.669} C_VEL
LIN {X 0,Y 601.424,Z 432.813,A -85,B 0,C 180,E1 -903.349,E2 -903.349} C_VEL
LIN {X 0,Y 601.426,Z 432.814,A -85,B 0,C 180,E1 -906.037,E2 -906.037} C_VEL
LIN {X 0,Y 601.435,Z 432.82,A -85,B 0,C 180,E1 -908.737,E2 -908.737} C_VEL
LIN {X 0,Y 601.426,Z 432.812,A -85,B 0,C 180,E1 -911.458,E2 -911.458} C_VEL
LIN {X 0,Y 601.406,Z 432.818,A -85,B 0,C 180,E1 -912.386,E2 -912.386} C_VEL
LIN {X 0,Y 600.74,Z 432.907,A -85,B 0,C 180,E1 -912.946,E2 -912.946} C_VEL
LIN {X 0,Y 597.887,Z 433.262,A -85,B 0,C 180,E1 -913.853,E2 -913.853} C_VEL
LIN {X 0,Y 595.476,Z 433.562,A -85,B 0,C 180,E1 -914.583,E2 -914.583} C_VEL
LIN {X 0,Y 594.439,Z 433.686,A -85,B 0,C 180,E1 -915.147,E2 -915.147} C_VEL
LIN {X 0,Y 594.354,Z 433.694,A -85,B 0,C 180,E1 -915.338,E2 -915.338} C_VEL
LIN {X 0,Y 594.374,Z 433.691,A -85,B 0,C 180,E1 -917.904,E2 -917.904} C_VEL
LIN {X 0,Y 594.374,Z 433.7,A -85,B 0,C 180,E1 -920.918,E2 -920.918} C_VEL
LIN {X 0,Y 594.386,Z 433.689,A -85,B 0,C 180,E1 -923.704,E2 -923.704} C_VEL
LIN {X 0,Y 594.38,Z 433.694,A -85,B 0,C 180,E1 -926.699,E2 -926.699} C_VEL
LIN {X 0,Y 594.373,Z 433.701,A -85,B 0,C 180,E1 -928.999,E2 -928.999} C_VEL
LIN {X 0,Y 594.383,Z 433.691,A -85,B 0,C 180,E1 -931.646,E2 -931.646} C_VEL
LIN {X 0,Y 594.385,Z 433.689,A -85,B 0,C 180,E1 -934.579,E2 -934.579} C_VEL
LIN {X 0,Y 594.38,Z 433.701,A -85,B 0,C 180,E1 -937.087,E2 -937.087} C_VEL
LIN {X 0,Y 594.37,Z 433.693,A -85,B 0,C 180,E1 -939.775,E2 -939.775} C_VEL
LIN {X 0,Y 594.366,Z 433.692,A -85,B 0,C 180,E1 -942.375,E2 -942.375} C_VEL
LIN {X 0,Y 594.355,Z 433.704,A -85,B 0,C 180,E1 -945.192,E2 -945.192} C_VEL
LIN {X 0,Y 594.361,Z 433.697,A -85,B 0,C 180,E1 -947.625,E2 -947.625} C_VEL
LIN {X 0,Y 594.386,Z 433.689,A -85,B 0,C 180,E1 -950.322,E2 -950.322} C_VEL
LIN {X 0,Y 594.378,Z 433.694,A -85,B 0,C 180,E1 -952.914,E2 -952.914} C_VEL
LIN {X 0,Y 594.381,Z 433.694,A -85,B 0,C 180,E1 -955.861,E2 -955.861} C_VEL
LIN {X 0,Y 594.384,Z 433.69,A -85,B 0,C 180,E1 -958.651,E2 -958.651} C_VEL
LIN {X 0,Y 594.38,Z 433.693,A -85,B 0,C 180,E1 -961.042,E2 -961.042} C_VEL
LIN {X 0,Y 594.384,Z 433.694,A -85,B 0,C 180,E1 -963.977,E2 -963.977} C_VEL
LIN {X 0,Y 594.385,Z 433.691,A -85,B 0,C 180,E1 -966.296,E2 -966.296} C_VEL
LIN {X 0,Y 594.4,Z 433.691,A -85,B 0,C 180,E1 -969.225,E2 -969.225} C_VEL
LIN {X 0,Y 594.376,Z 433.695,A -85,B 0,C 180,E1 -972.096,E2 -972.096} C_VEL
LIN {X 0,Y 594.365,Z 433.695,A -85,B 0,C 180,E1 -974.219,E2 -974.219} C_VEL
LIN {X 0,Y 594.368,Z 433.692,A -85,B 0,C 180,E1 -977.017,E2 -977.017} C_VEL
LIN {X 0,Y 594.386,Z 433.7,A -85,B 0,C 180,E1 -979.784,E2 -979.784} C_VEL
LIN {X 0,Y 594.4,Z 433.689,A -85,B 0,C 180,E1 -982.527,E2 -982.527} C_VEL
LIN {X 0,Y 594.385,Z 433.691,A -85,B 0,C 180,E1 -985.252,E2 -985.252} C_VEL
LIN {X 0,Y 594.4,Z 433.698,A -85,B 0,C 180,E1 -987.967,E2 -987.967} C_VEL
LIN {X 0,Y 594.413,Z 433.687,A -85,B 0,C 180,E1 -990.677,E2 -990.677} C_VEL
LIN {X 0,Y 594.38,Z 433.692,A -85,B 0,C 180,E1 -993.389,E2 -993.389} C_VEL
LIN {X 0,Y 594.363,Z 433.703,A -85,B 0,C 180,E1 -996.109,E2 -996.109} C_VEL
LIN {X 0,Y 594.379,Z 433.691,A -85,B 0,C 180,E1 -998.842,E2 -998.842} C_VEL
LIN {X 0,Y 594.392,Z 433.691,A -85,B 0,C 180,E1 -1001.595,E2 -1001.595} C_VEL
LIN {X 0,Y 594.385,Z 433.698,A -85,B 0,C 180,E1 -1004.377,E2 -1004.377} C_VEL
LIN {X 0,Y 594.389,Z 433.689,A -85,B 0,C 180,E1 -1007.193,E2 -1007.193} C_VEL
LIN {X 0,Y 594.372,Z 433.697,A -85,B 0,C 180,E1 -1010.053,E2 -1010.053} C_VEL
LIN {X 0,Y 594.359,Z 433.695,A -85,B 0,C 180,E1 -1012.967,E2 -1012.967} C_VEL
LIN {X 0,Y 594.372,Z 433.692,A -85,B 0,C 180,E1 -1015.193,E2 -1015.193} C_VEL
LIN {X 0,Y 594.38,Z 433.69,A -85,B 0,C 180,E1 -1017.526,E2 -1017.526} C_VEL
LIN {X 0,Y 594.38,Z 433.698,A -85,B 0,C 180,E1 -1020.328,E2 -1020.328} C_VEL
LIN {X 0,Y 594.374,Z 433.695,A -85,B 0,C 180,E1 -1022.95,E2 -1022.95} C_VEL
LIN {X 0,Y 594.378,Z 433.691,A -85,B 0,C 180,E1 -1025.406,E2 -1025.406} C_VEL
LIN {X 0,Y 594.378,Z 433.691,A -85,B 0,C 180,E1 -1027.94,E2 -1027.94} C_VEL
LIN {X 0,Y 594.371,Z 433.7,A -85,B 0,C 180,E1 -1030.822,E2 -1030.822} C_VEL
LIN {X 0,Y 594.373,Z 433.691,A -85,B 0,C 180,E1 -1033.841,E2 -1033.841} C_VEL
LIN {X 0,Y 594.373,Z 433.701,A -85,B 0,C 180,E1 -1036.702,E2 -1036.702} C_VEL
LIN {X 0,Y 594.381,Z 433.692,A -85,B 0,C 180,E1 -1039.435,E2 -1039.435} C_VEL
LIN {X 0,Y 594.384,Z 433.693,A -85,B 0,C 180,E1 -1042.391,E2 -1042.391} C_VEL
LIN {X 0,Y 594.375,Z 433.697,A -85,B 0,C 180,E1 -1044.671,E2 -1044.671} C_VEL
LIN {X 0,Y 594.369,Z 433.699,A -85,B 0,C 180,E1 -1047.088,E2 -1047.088} C_VEL
LIN {X 0,Y 594.391,Z 433.69,A -85,B 0,C 180,E1 -1049.669,E2 -1049.669} C_VEL
LIN {X 0,Y 594.381,Z 433.691,A -85,B 0,C 180,E1 -1052.54,E2 -1052.54} C_VEL
LIN {X 0,Y 594.37,Z 433.694,A -85,B 0,C 180,E1 -1054.807,E2 -1054.807} C_VEL
LIN {X 0,Y 594.355,Z 433.702,A -85,B 0,C 180,E1 -1057.264,E2 -1057.264} C_VEL
LIN {X 0,Y 594.369,Z 433.691,A -85,B 0,C 180,E1 -1059.946,E2 -1059.946} C_VEL
LIN {X 0,Y 594.382,Z 433.694,A -85,B 0,C 180,E1 -1062.807,E2 -1062.807} C_VEL
LIN {X 0,Y 594.378,Z 433.692,A -85,B 0,C 180,E1 -1065.826,E2 -1065.826} C_VEL
LIN {X 0,Y 594.386,Z 433.688,A -85,B 0,C 180,E1 -1068.404,E2 -1068.404} C_VEL
LIN {X 0,Y 594.395,Z 433.695,A -85,B 0,C 180,E1 -1071.158,E2 -1071.158} C_VEL
LIN {X 0,Y 594.38,Z 433.692,A -85,B 0,C 180,E1 -1073.891,E2 -1073.891} C_VEL
LIN {X 0,Y 594.376,Z 433.691,A -85,B 0,C 180,E1 -1076.611,E2 -1076.611} C_VEL
LIN {X 0,Y 594.416,Z 433.692,A -85,B 0,C 180,E1 -1079.323,E2 -1079.323} C_VEL
LIN {X 0,Y 594.387,Z 433.692,A -85,B 0,C 180,E1 -1082.033,E2 -1082.033} C_VEL
LIN {X 0,Y 594.399,Z 433.687,A -85,B 0,C 180,E1 -1084.748,E2 -1084.748} C_VEL
LIN {X 0,Y 594.385,Z 433.697,A -85,B 0,C 180,E1 -1087.473,E2 -1087.473} C_VEL
LIN {X 0,Y 594.391,Z 433.691,A -85,B 0,C 180,E1 -1090.216,E2 -1090.216} C_VEL
LIN {X 0,Y 594.362,Z 433.692,A -85,B 0,C 180,E1 -1092.983,E2 -1092.983} C_VEL
LIN {X 0,Y 594.362,Z 433.703,A -85,B 0,C 180,E1 -1095.781,E2 -1095.781} C_VEL
LIN {X 0,Y 594.38,Z 433.688,A -85,B 0,C 180,E1 -1098.618,E2 -1098.618} C_VEL
LIN {X 0,Y 594.36,Z 433.694,A -85,B 0,C 180,E1 -1101.504,E2 -1101.504} C_VEL
LIN {X 0,Y 594.38,Z 433.693,A -85,B 0,C 180,E1 -1104.446,E2 -1104.446} C_VEL
LIN {X 0,Y 594.38,Z 433.689,A -85,B 0,C 180,E1 -1106.7,E2 -1106.7} C_VEL
LIN {X 0,Y 594.373,Z 433.688,A -85,B 0,C 180,E1 -1108.999,E2 -1108.999} C_VEL
LIN {X 0,Y 594.384,Z 433.693,A -85,B 0,C 180,E1 -1111.646,E2 -1111.646} C_VEL
LIN {X 0,Y 594.386,Z 433.69,A -85,B 0,C 180,E1 -1114.579,E2 -1114.579} C_VEL
LIN {X 0,Y 594.382,Z 433.69,A -85,B 0,C 180,E1 -1117.087,E2 -1117.087} C_VEL
LIN {X 0,Y 594.371,Z 433.694,A -85,B 0,C 180,E1 -1119.775,E2 -1119.775} C_VEL
LIN {X 0,Y 594.367,Z 433.7,A -85,B 0,C 180,E1 -1122.375,E2 -1122.375} C_VEL
LIN {X 0,Y 594.356,Z 433.693,A -85,B 0,C 180,E1 -1125.192,E2 -1125.192} C_VEL
LIN {X 0,Y 594.376,Z 433.698,A -85,B 0,C 180,E1 -1128.152,E2 -1128.152} C_VEL
LIN {X 0,Y 594.381,Z 433.688,A -85,B 0,C 180,E1 -1131.196,E2 -1131.196} C_VEL
LIN {X 0,Y 594.391,Z 433.69,A -85,B 0,C 180,E1 -1133.759,E2 -1133.759} C_VEL
LIN {X 0,Y 594.378,Z 433.696,A -85,B 0,C 180,E1 -1136.24,E2 -1136.24} C_VEL
LIN {X 0,Y 594.386,Z 433.692,A -85,B 0,C 180,E1 -1138.651,E2 -1138.651} C_VEL
LIN {X 0,Y 594.421,Z 433.883,A -85,B 0,C 180,E1 -1139.876,E2 -1139.876} C_VEL
LIN {X 0,Y 595.277,Z 437.776,A -85,B 0,C 180,E1 -1140.46,E2 -1140.46} C_VEL
LIN {X 0,Y 595.14,Z 457.291,A -85,B 0,C 180,E1 -1142.959,E2 -1142.959} C_VEL
LIN {X 0,Y 594.995,Z 478.235,A -85,B 0,C 180,E1 -1145.581,E2 -1145.581} C_VEL
LIN {X 0,Y 595.003,Z 484.411,A -85,B 0,C 180,E1 -1146.311,E2 -1146.311} C_VEL
LIN {X 0,Y 595.938,Z 488.609,A -85,B 0,C 180,E1 -1146.418,E2 -1146.418} C_VEL
LIN {X 0,Y 595.542,Z 696.305,A -85,B 0,C 180,E1 -1149.072,E2 -1149.072} C_VEL
LIN {X 0,Y 595.47,Z 713.153,A -85,B 0,C 180,E1 -1149.422,E2 -1149.422} C_VEL
LIN {X 0,Y 595.362,Z 730.585,A -85,B 0,C 180,E1 -1149.936,E2 -1149.936} C_VEL
LIN {X 0,Y 595.216,Z 746.779,A -85,B 0,C 180,E1 -1150.56,E2 -1150.56} C_VEL
LIN {X 0,Y 595.09,Z 763.156,A -85,B 0,C 180,E1 -1151.353,E2 -1151.353} C_VEL
LIN {X 0,Y 594.937,Z 778.99,A -85,B 0,C 180,E1 -1152.291,E2 -1152.291} C_VEL
LIN {X 0,Y 594.791,Z 793.174,A -85,B 0,C 180,E1 -1153.3,E2 -1153.3} C_VEL
LIN {X 0,Y 594.654,Z 806.426,A -85,B 0,C 180,E1 -1154.403,E2 -1154.403} C_VEL
LIN {X 0,Y 594.554,Z 818.984,A -85,B 0,C 180,E1 -1155.627,E2 -1155.627} C_VEL
LIN {X 0,Y 594.464,Z 829.723,A -85,B 0,C 180,E1 -1156.846,E2 -1156.846} C_VEL
LIN {X 0,Y 594.404,Z 840.146,A -85,B 0,C 180,E1 -1158.232,E2 -1158.232} C_VEL
LIN {X 0,Y 594.355,Z 848.903,A -85,B 0,C 180,E1 -1159.612,E2 -1159.612} C_VEL
LIN {X 0,Y 594.298,Z 857.129,A -85,B 0,C 180,E1 -1161.157,E2 -1161.157} C_VEL
LIN {X 0,Y 594.281,Z 863.147,A -85,B 0,C 180,E1 -1162.526,E2 -1162.526} C_VEL
LIN {X 0,Y 594.25,Z 867.957,A -85,B 0,C 180,E1 -1163.89,E2 -1163.89} C_VEL
LIN {X 0,Y 594.223,Z 871.796,A -85,B 0,C 180,E1 -1165.251,E2 -1165.251} C_VEL
LIN {X 0,Y 594.256,Z 874.568,A -85,B 0,C 180,E1 -1166.61,E2 -1166.61} C_VEL
LIN {X 0,Y 594.235,Z 876.436,A -85,B 0,C 180,E1 -1167.967,E2 -1167.967} C_VEL
LIN {X 0,Y 594.235,Z 877.35,A -85,B 0,C 180,E1 -1169.322,E2 -1169.322} C_VEL
LIN {X 0,Y 594.235,Z 877.35,A -85,B 0,C 180,E1 -1170.678,E2 -1170.678} C_VEL
LIN {X 0,Y 594.235,Z 876.436,A -85,B 0,C 180,E1 -1172.033,E2 -1172.033} C_VEL
LIN {X 0,Y 594.256,Z 874.568,A -85,B 0,C 180,E1 -1173.39,E2 -1173.39} C_VEL
LIN {X 0,Y 594.223,Z 871.796,A -85,B 0,C 180,E1 -1174.749,E2 -1174.749} C_VEL
LIN {X 0,Y 594.25,Z 867.957,A -85,B 0,C 180,E1 -1176.11,E2 -1176.11} C_VEL
LIN {X 0,Y 594.281,Z 863.147,A -85,B 0,C 180,E1 -1177.474,E2 -1177.474} C_VEL
LIN {X 0,Y 594.298,Z 857.129,A -85,B 0,C 180,E1 -1178.843,E2 -1178.843} C_VEL
LIN {X 0,Y 594.355,Z 848.903,A -85,B 0,C 180,E1 -1180.388,E2 -1180.388} C_VEL
LIN {X 0,Y 594.404,Z 840.146,A -85,B 0,C 180,E1 -1181.768,E2 -1181.768} C_VEL
LIN {X 0,Y 594.464,Z 829.723,A -85,B 0,C 180,E1 -1183.154,E2 -1183.154} C_VEL
LIN {X 0,Y 594.563,Z 817.356,A -85,B 0,C 180,E1 -1184.547,E2 -1184.547} C_VEL
LIN {X 0,Y 594.677,Z 804.486,A -85,B 0,C 180,E1 -1185.772,E2 -1185.772} C_VEL
LIN {X 0,Y 594.806,Z 791.184,A -85,B 0,C 180,E1 -1186.851,E2 -1186.851} C_VEL
LIN {X 0,Y 594.958,Z 776.168,A -85,B 0,C 180,E1 -1187.886,E2 -1187.886} C_VEL
LIN {X 0,Y 595.117,Z 761.092,A -85,B 0,C 180,E1 -1188.753,E2 -1188.753} C_VEL
LIN {X 0,Y 595.227,Z 744.732,A -85,B 0,C 180,E1 -1189.529,E2 -1189.529} C_VEL
LIN {X 0,Y 595.368,Z 728,A -85,B 0,C 180,E1 -1190.153,E2 -1190.153} C_VEL
LIN {X 0,Y 595.471,Z 711.327,A -85,B 0,C 180,E1 -1190.623,E2 -1190.623} C_VEL
LIN {X 0,Y 595.537,Z 695.049,A -85,B 0,C 180,E1 -1190.947,E2 -1190.947} C_VEL
LIN {X 0,Y 595.906,Z 488.698,A -85,B 0,C 180,E1 -1193.582,E2 -1193.582} C_VEL
LIN {X 0,Y 594.991,Z 484.215,A -85,B 0,C 180,E1 -1193.701,E2 -1193.701} C_VEL
LIN {X 0,Y 595.098,Z 462.798,A -85,B 0,C 180,E1 -1196.347,E2 -1196.347} C_VEL
LIN {X 0,Y 595.348,Z 439.21,A -85,B 0,C 180,E1 -1199.35,E2 -1199.35} C_VEL
LIN {X 0,Y 594.432,Z 433.946,A -85,B 0,C 180,E1 -1200.101,E2 -1200.101} C_VEL
LIN {X 0,Y 594.382,Z 433.684,A -85,B 0,C 180,E1 -1200.559,E2 -1200.559} C_VEL
LIN {X 0,Y 594.376,Z 433.695,A -85,B 0,C 180,E1 -1202.949,E2 -1202.949} C_VEL
LIN {X 0,Y 594.38,Z 433.697,A -85,B 0,C 180,E1 -1205.406,E2 -1205.406} C_VEL
LIN {X 0,Y 594.379,Z 433.693,A -85,B 0,C 180,E1 -1207.94,E2 -1207.94} C_VEL
LIN {X 0,Y 594.371,Z 433.692,A -85,B 0,C 180,E1 -1210.822,E2 -1210.822} C_VEL
LIN {X 0,Y 594.36,Z 433.696,A -85,B 0,C 180,E1 -1213.299,E2 -1213.299} C_VEL
LIN {X 0,Y 594.376,Z 433.694,A -85,B 0,C 180,E1 -1216.158,E2 -1216.158} C_VEL
LIN {X 0,Y 594.384,Z 433.691,A -85,B 0,C 180,E1 -1219.176,E2 -1219.176} C_VEL
LIN {X 0,Y 594.384,Z 433.697,A -85,B 0,C 180,E1 -1222.059,E2 -1222.059} C_VEL
LIN {X 0,Y 594.376,Z 433.689,A -85,B 0,C 180,E1 -1224.671,E2 -1224.671} C_VEL
LIN {X 0,Y 594.371,Z 433.691,A -85,B 0,C 180,E1 -1227.088,E2 -1227.088} C_VEL
LIN {X 0,Y 594.393,Z 433.694,A -85,B 0,C 180,E1 -1229.669,E2 -1229.669} C_VEL
LIN {X 0,Y 594.365,Z 433.693,A -85,B 0,C 180,E1 -1232.539,E2 -1232.539} C_VEL
LIN {X 0,Y 594.371,Z 433.692,A -85,B 0,C 180,E1 -1234.807,E2 -1234.807} C_VEL
LIN {X 0,Y 594.356,Z 433.693,A -85,B 0,C 180,E1 -1237.264,E2 -1237.264} C_VEL
LIN {X 0,Y 594.369,Z 433.695,A -85,B 0,C 180,E1 -1239.946,E2 -1239.946} C_VEL
LIN {X 0,Y 594.383,Z 433.691,A -85,B 0,C 180,E1 -1242.806,E2 -1242.806} C_VEL
LIN {X 0,Y 594.379,Z 433.694,A -85,B 0,C 180,E1 -1245.825,E2 -1245.825} C_VEL
LIN {X 0,Y 594.386,Z 433.698,A -85,B 0,C 180,E1 -1248.404,E2 -1248.404} C_VEL
LIN {X 0,Y 594.394,Z 433.687,A -85,B 0,C 180,E1 -1251.158,E2 -1251.158} C_VEL
LIN {X 0,Y 594.362,Z 433.695,A -85,B 0,C 180,E1 -1253.891,E2 -1253.891} C_VEL
LIN {X 0,Y 594.376,Z 433.698,A -85,B 0,C 180,E1 -1256.611,E2 -1256.611} C_VEL
LIN {X 0,Y 594.418,Z 433.685,A -85,B 0,C 180,E1 -1259.322,E2 -1259.322} C_VEL
LIN {X 0,Y 594.387,Z 433.691,A -85,B 0,C 180,E1 -1262.033,E2 -1262.033} C_VEL
LIN {X 0,Y 594.398,Z 433.695,A -85,B 0,C 180,E1 -1264.747,E2 -1264.747} C_VEL
LIN {X 0,Y 594.385,Z 433.689,A -85,B 0,C 180,E1 -1267.473,E2 -1267.473} C_VEL
LIN {X 0,Y 594.39,Z 433.692,A -85,B 0,C 180,E1 -1270.216,E2 -1270.216} C_VEL
LIN {X 0,Y 594.363,Z 433.698,A -85,B 0,C 180,E1 -1272.983,E2 -1272.983} C_VEL
LIN {X 0,Y 594.354,Z 433.694,A -85,B 0,C 180,E1 -1275.338,E2 -1275.338} C_VEL
LIN {X 0,Y 593.685,Z 433.778,A -85,B 0,C 180,E1 -1275.904,E2 -1275.904} C_VEL
LIN {X 0,Y 590.832,Z 434.142,A -85,B 0,C 180,E1 -1276.822,E2 -1276.822} C_VEL
LIN {X 0,Y 588.427,Z 434.437,A -85,B 0,C 180,E1 -1277.561,E2 -1277.561} C_VEL
LIN {X 0,Y 587.399,Z 434.561,A -85,B 0,C 180,E1 -1278.131,E2 -1278.131} C_VEL
LIN {X 0,Y 587.318,Z 434.572,A -85,B 0,C 180,E1 -1278.324,E2 -1278.324} C_VEL
LIN {X 0,Y 587.348,Z 434.573,A -85,B 0,C 180,E1 -1281.045,E2 -1281.045} C_VEL
LIN {X 0,Y 587.33,Z 434.568,A -85,B 0,C 180,E1 -1284.006,E2 -1284.006} C_VEL
LIN {X 0,Y 587.353,Z 434.563,A -85,B 0,C 180,E1 -1286.278,E2 -1286.278} C_VEL
LIN {X 0,Y 587.342,Z 434.575,A -85,B 0,C 180,E1 -1289.134,E2 -1289.134} C_VEL
LIN {X 0,Y 587.346,Z 434.566,A -85,B 0,C 180,E1 -1291.838,E2 -1291.838} C_VEL
LIN {X 0,Y 587.346,Z 434.562,A -85,B 0,C 180,E1 -1294.349,E2 -1294.349} C_VEL
LIN {X 0,Y 587.345,Z 434.571,A -85,B 0,C 180,E1 -1296.747,E2 -1296.747} C_VEL
LIN {X 0,Y 587.34,Z 434.574,A -85,B 0,C 180,E1 -1299.359,E2 -1299.359} C_VEL
LIN {X 0,Y 587.325,Z 434.569,A -85,B 0,C 180,E1 -1302.108,E2 -1302.108} C_VEL
LIN {X 0,Y 587.308,Z 434.579,A -85,B 0,C 180,E1 -1305.089,E2 -1305.089} C_VEL
LIN {X 0,Y 587.345,Z 434.568,A -85,B 0,C 180,E1 -1307.928,E2 -1307.928} C_VEL
LIN {X 0,Y 587.327,Z 434.575,A -85,B 0,C 180,E1 -1311.058,E2 -1311.058} C_VEL
LIN {X 0,Y 587.347,Z 434.576,A -85,B 0,C 180,E1 -1313.292,E2 -1313.292} C_VEL
LIN {X 0,Y 587.363,Z 434.569,A -85,B 0,C 180,E1 -1315.781,E2 -1315.781} C_VEL
LIN {X 0,Y 587.348,Z 434.567,A -85,B 0,C 180,E1 -1318.232,E2 -1318.232} C_VEL
LIN {X 0,Y 587.345,Z 434.568,A -85,B 0,C 180,E1 -1320.866,E2 -1320.866} C_VEL
LIN {X 0,Y 587.355,Z 434.572,A -85,B 0,C 180,E1 -1323.819,E2 -1323.819} C_VEL
LIN {X 0,Y 587.332,Z 434.573,A -85,B 0,C 180,E1 -1325.994,E2 -1325.994} C_VEL
LIN {X 0,Y 587.32,Z 434.572,A -85,B 0,C 180,E1 -1328.226,E2 -1328.226} C_VEL
LIN {X 0,Y 587.344,Z 434.57,A -85,B 0,C 180,E1 -1331.152,E2 -1331.152} C_VEL
LIN {X 0,Y 587.348,Z 434.57,A -85,B 0,C 180,E1 -1333.311,E2 -1333.311} C_VEL
LIN {X 0,Y 587.359,Z 434.569,A -85,B 0,C 180,E1 -1336.155,E2 -1336.155} C_VEL
LIN {X 0,Y 587.336,Z 434.568,A -85,B 0,C 180,E1 -1338.963,E2 -1338.963} C_VEL
LIN {X 0,Y 587.361,Z 434.574,A -85,B 0,C 180,E1 -1341.745,E2 -1341.745} C_VEL
LIN {X 0,Y 587.355,Z 434.567,A -85,B 0,C 180,E1 -1344.507,E2 -1344.507} C_VEL
LIN {X 0,Y 587.368,Z 434.565,A -85,B 0,C 180,E1 -1347.257,E2 -1347.257} C_VEL
LIN {X 0,Y 587.382,Z 434.573,A -85,B 0,C 180,E1 -1350,E2 -1350} C_VEL
LIN {X 0,Y 587.368,Z 434.565,A -85,B 0,C 180,E1 -1352.743,E2 -1352.743} C_VEL
LIN {X 0,Y 587.355,Z 434.567,A -85,B 0,C 180,E1 -1355.493,E2 -1355.493} C_VEL
LIN {X 0,Y 587.361,Z 434.574,A -85,B 0,C 180,E1 -1358.255,E2 -1358.255} C_VEL
LIN {X 0,Y 587.344,Z 434.567,A -85,B 0,C 180,E1 -1361.133,E2 -1361.133} C_VEL
LIN {X 0,Y 587.361,Z 434.575,A -85,B 0,C 180,E1 -1364.26,E2 -1364.26} C_VEL
LIN {X 0,Y 587.355,Z 434.565,A -85,B 0,C 180,E1 -1367.405,E2 -1367.405} C_VEL
LIN {X 0,Y 587.327,Z 434.579,A -85,B 0,C 180,E1 -1370.304,E2 -1370.304} C_VEL
LIN {X 0,Y 587.317,Z 434.57,A -85,B 0,C 180,E1 -1373.258,E2 -1373.258} C_VEL
LIN {X 0,Y 587.332,Z 434.568,A -85,B 0,C 180,E1 -1375.516,E2 -1375.516} C_VEL
LIN {X 0,Y 587.344,Z 434.568,A -85,B 0,C 180,E1 -1377.817,E2 -1377.817} C_VEL
LIN {X 0,Y 587.335,Z 434.579,A -85,B 0,C 180,E1 -1380.51,E2 -1380.51} C_VEL
LIN {X 0,Y 587.335,Z 434.57,A -85,B 0,C 180,E1 -1383.112,E2 -1383.112} C_VEL
LIN {X 0,Y 587.35,Z 434.567,A -85,B 0,C 180,E1 -1385.895,E2 -1385.895} C_VEL
LIN {X 0,Y 587.325,Z 434.577,A -85,B 0,C 180,E1 -1388.479,E2 -1388.479} C_VEL
LIN {X 0,Y 587.329,Z 434.572,A -85,B 0,C 180,E1 -1391.156,E2 -1391.156} C_VEL
LIN {X 0,Y 587.325,Z 434.571,A -85,B 0,C 180,E1 -1394.114,E2 -1394.114} C_VEL
LIN {X 0,Y 587.316,Z 434.577,A -85,B 0,C 180,E1 -1396.994,E2 -1396.994} C_VEL
LIN {X 0,Y 587.321,Z 434.57,A -85,B 0,C 180,E1 -1399.747,E2 -1399.747} C_VEL
LIN {X 0,Y 587.339,Z 434.57,A -85,B 0,C 180,E1 -1402.392,E2 -1402.392} C_VEL
LIN {X 0,Y 587.34,Z 434.573,A -85,B 0,C 180,E1 -1404.946,E2 -1404.946} C_VEL
LIN {X 0,Y 587.331,Z 434.571,A -85,B 0,C 180,E1 -1407.421,E2 -1407.421} C_VEL
LIN {X 0,Y 587.338,Z 434.568,A -85,B 0,C 180,E1 -1409.831,E2 -1409.831} C_VEL
LIN {X 0,Y 587.341,Z 434.565,A -85,B 0,C 180,E1 -1412.307,E2 -1412.307} C_VEL
LIN {X 0,Y 587.329,Z 434.566,A -85,B 0,C 180,E1 -1414.483,E2 -1414.483} C_VEL
LIN {X 0,Y 587.31,Z 434.582,A -85,B 0,C 180,E1 -1417.131,E2 -1417.131} C_VEL
LIN {X 0,Y 587.324,Z 434.571,A -85,B 0,C 180,E1 -1419.695,E2 -1419.695} C_VEL
LIN {X 0,Y 587.35,Z 434.567,A -85,B 0,C 180,E1 -1422.594,E2 -1422.594} C_VEL
LIN {X 0,Y 587.354,Z 434.568,A -85,B 0,C 180,E1 -1425.739,E2 -1425.739} C_VEL
LIN {X 0,Y 587.352,Z 434.567,A -85,B 0,C 180,E1 -1428.859,E2 -1428.859} C_VEL
LIN {X 0,Y 587.365,Z 434.568,A -85,B 0,C 180,E1 -1431.745,E2 -1431.745} C_VEL
LIN {X 0,Y 587.355,Z 434.564,A -85,B 0,C 180,E1 -1434.507,E2 -1434.507} C_VEL
LIN {X 0,Y 587.374,Z 434.57,A -85,B 0,C 180,E1 -1437.257,E2 -1437.257} C_VEL
LIN {X 0,Y 587.373,Z 434.566,A -85,B 0,C 180,E1 -1440,E2 -1440} C_VEL
LIN {X 0,Y 587.375,Z 434.562,A -85,B 0,C 180,E1 -1442.743,E2 -1442.743} C_VEL
LIN {X 0,Y 587.349,Z 434.574,A -85,B 0,C 180,E1 -1445.493,E2 -1445.493} C_VEL
LIN {X 0,Y 587.365,Z 434.564,A -85,B 0,C 180,E1 -1448.255,E2 -1448.255} C_VEL
LIN {X 0,Y 587.352,Z 434.567,A -85,B 0,C 180,E1 -1451.142,E2 -1451.142} C_VEL
LIN {X 0,Y 587.355,Z 434.567,A -85,B 0,C 180,E1 -1454.261,E2 -1454.261} C_VEL
LIN {X 0,Y 587.35,Z 434.569,A -85,B 0,C 180,E1 -1457.406,E2 -1457.406} C_VEL
LIN {X 0,Y 587.324,Z 434.568,A -85,B 0,C 180,E1 -1460.305,E2 -1460.305} C_VEL
LIN {X 0,Y 587.316,Z 434.571,A -85,B 0,C 180,E1 -1463.259,E2 -1463.259} C_VEL
LIN {X 0,Y 587.329,Z 434.572,A -85,B 0,C 180,E1 -1465.517,E2 -1465.517} C_VEL
LIN {X 0,Y 587.34,Z 434.573,A -85,B 0,C 180,E1 -1467.818,E2 -1467.818} C_VEL
LIN {X 0,Y 587.344,Z 434.569,A -85,B 0,C 180,E1 -1470.513,E2 -1470.513} C_VEL
LIN {X 0,Y 587.328,Z 434.569,A -85,B 0,C 180,E1 -1473.397,E2 -1473.397} C_VEL
LIN {X 0,Y 587.348,Z 434.57,A -85,B 0,C 180,E1 -1475.896,E2 -1475.896} C_VEL
LIN {X 0,Y 587.33,Z 434.573,A -85,B 0,C 180,E1 -1478.479,E2 -1478.479} C_VEL
LIN {X 0,Y 587.334,Z 434.567,A -85,B 0,C 180,E1 -1481.157,E2 -1481.157} C_VEL
LIN {X 0,Y 587.328,Z 434.577,A -85,B 0,C 180,E1 -1484.115,E2 -1484.115} C_VEL
LIN {X 0,Y 587.308,Z 434.571,A -85,B 0,C 180,E1 -1486.994,E2 -1486.994} C_VEL
LIN {X 0,Y 587.313,Z 434.573,A -85,B 0,C 180,E1 -1489.747,E2 -1489.747} C_VEL
LIN {X 0,Y 587.339,Z 434.571,A -85,B 0,C 180,E1 -1492.393,E2 -1492.393} C_VEL
LIN {X 0,Y 587.346,Z 434.568,A -85,B 0,C 180,E1 -1494.947,E2 -1494.947} C_VEL
LIN {X 0,Y 587.338,Z 434.571,A -85,B 0,C 180,E1 -1497.422,E2 -1497.422} C_VEL
LIN {X 0,Y 587.38,Z 434.724,A -85,B 0,C 180,E1 -1499.586,E2 -1499.586} C_VEL
LIN {X 0,Y 588.546,Z 439.639,A -85,B 0,C 180,E1 -1500.333,E2 -1500.333} C_VEL
LIN {X 0,Y 588.37,Z 458.787,A -85,B 0,C 180,E1 -1502.814,E2 -1502.814} C_VEL
LIN {X 0,Y 588.151,Z 480.11,A -85,B 0,C 180,E1 -1505.514,E2 -1505.514} C_VEL
LIN {X 0,Y 588.192,Z 484.436,A -85,B 0,C 180,E1 -1506.02,E2 -1506.02} C_VEL
LIN {X 0,Y 589.417,Z 490.339,A -85,B 0,C 180,E1 -1506.164,E2 -1506.164} C_VEL
LIN {X 0,Y 588.917,Z 695.939,A -85,B 0,C 180,E1 -1508.82,E2 -1508.82} C_VEL
LIN {X 0,Y 588.81,Z 712.25,A -85,B 0,C 180,E1 -1509.156,E2 -1509.156} C_VEL
LIN {X 0,Y 588.652,Z 729.297,A -85,B 0,C 180,E1 -1509.652,E2 -1509.652} C_VEL
LIN {X 0,Y 588.484,Z 745.742,A -85,B 0,C 180,E1 -1510.283,E2 -1510.283} C_VEL
LIN {X 0,Y 588.323,Z 760.453,A -85,B 0,C 180,E1 -1510.99,E2 -1510.99} C_VEL
LIN {X 0,Y 588.154,Z 774.762,A -85,B 0,C 180,E1 -1511.81,E2 -1511.81} C_VEL
LIN {X 0,Y 587.952,Z 788.637,A -85,B 0,C 180,E1 -1512.75,E2 -1512.75} C_VEL
LIN {X 0,Y 587.757,Z 802.483,A -85,B 0,C 180,E1 -1513.859,E2 -1513.859} C_VEL
LIN {X 0,Y 587.61,Z 813.834,A -85,B 0,C 180,E1 -1514.922,E2 -1514.922} C_VEL
LIN {X 0,Y 587.534,Z 825.305,A -85,B 0,C 180,E1 -1516.159,E2 -1516.159} C_VEL
LIN {X 0,Y 587.393,Z 836.433,A -85,B 0,C 180,E1 -1517.563,E2 -1517.563} C_VEL
LIN {X 0,Y 587.335,Z 845.828,A -85,B 0,C 180,E1 -1518.963,E2 -1518.963} C_VEL
LIN {X 0,Y 587.244,Z 853.667,A -85,B 0,C 180,E1 -1520.355,E2 -1520.355} C_VEL
LIN {X 0,Y 587.226,Z 860.298,A -85,B 0,C 180,E1 -1521.743,E2 -1521.743} C_VEL
LIN {X 0,Y 587.189,Z 866.722,A -85,B 0,C 180,E1 -1523.42,E2 -1523.42} C_VEL
LIN {X 0,Y 587.189,Z 870.021,A -85,B 0,C 180,E1 -1524.506,E2 -1524.506} C_VEL
LIN {X 0,Y 587.165,Z 873.291,A -85,B 0,C 180,E1 -1525.882,E2 -1525.882} C_VEL
LIN {X 0,Y 587.123,Z 875.654,A -85,B 0,C 180,E1 -1527.256,E2 -1527.256} C_VEL
LIN {X 0,Y 587.14,Z 876.999,A -85,B 0,C 180,E1 -1528.628,E2 -1528.628} C_VEL
LIN {X 0,Y 587.131,Z 877.5,A -85,B 0,C 180,E1 -1530,E2 -1530} C_VEL
LIN {X 0,Y 587.14,Z 876.999,A -85,B 0,C 180,E1 -1531.372,E2 -1531.372} C_VEL
LIN {X 0,Y 587.123,Z 875.654,A -85,B 0,C 180,E1 -1532.744,E2 -1532.744} C_VEL
LIN {X 0,Y 587.164,Z 873.291,A -85,B 0,C 180,E1 -1534.118,E2 -1534.118} C_VEL
LIN {X 0,Y 587.189,Z 870.021,A -85,B 0,C 180,E1 -1535.494,E2 -1535.494} C_VEL
LIN {X 0,Y 587.203,Z 865.668,A -85,B 0,C 180,E1 -1536.874,E2 -1536.874} C_VEL
LIN {X 0,Y 587.226,Z 860.298,A -85,B 0,C 180,E1 -1538.257,E2 -1538.257} C_VEL
LIN {X 0,Y 587.244,Z 853.667,A -85,B 0,C 180,E1 -1539.645,E2 -1539.645} C_VEL
LIN {X 0,Y 587.328,Z 845.283,A -85,B 0,C 180,E1 -1541.124,E2 -1541.124} C_VEL
LIN {X 0,Y 587.403,Z 835.169,A -85,B 0,C 180,E1 -1542.612,E2 -1542.612} C_VEL
LIN {X 0,Y 587.524,Z 823.823,A -85,B 0,C 180,E1 -1544.015,E2 -1544.015} C_VEL
LIN {X 0,Y 587.672,Z 812.057,A -85,B 0,C 180,E1 -1545.254,E2 -1545.254} C_VEL
LIN {X 0,Y 587.809,Z 799.32,A -85,B 0,C 180,E1 -1546.407,E2 -1546.407} C_VEL
LIN {X 0,Y 587.998,Z 785.462,A -85,B 0,C 180,E1 -1547.475,E2 -1547.475} C_VEL
LIN {X 0,Y 588.178,Z 771.873,A -85,B 0,C 180,E1 -1548.369,E2 -1548.369} C_VEL
LIN {X 0,Y 588.36,Z 757.412,A -85,B 0,C 180,E1 -1549.167,E2 -1549.167} C_VEL
LIN {X 0,Y 588.554,Z 741.418,A -85,B 0,C 180,E1 -1549.896,E2 -1549.896} C_VEL
LIN {X 0,Y 588.713,Z 724.393,A -85,B 0,C 180,E1 -1550.505,E2 -1550.505} C_VEL
LIN {X 0,Y 588.858,Z 708.502,A -85,B 0,C 180,E1 -1550.934,E2 -1550.934} C_VEL
LIN {X 0,Y 588.924,Z 692.121,A -85,B 0,C 180,E1 -1551.238,E2 -1551.238} C_VEL
LIN {X 0,Y 589.398,Z 493.077,A -85,B 0,C 180,E1 -1553.801,E2 -1553.801} C_VEL
LIN {X 0,Y 589.198,Z 488.651,A -85,B 0,C 180,E1 -1553.867,E2 -1553.867} C_VEL
LIN {X 0,Y 588.175,Z 484.226,A -85,B 0,C 180,E1 -1553.993,E2 -1553.993} C_VEL
LIN {X 0,Y 588.355,Z 463.259,A -85,B 0,C 180,E1 -1556.613,E2 -1556.613} C_VEL
LIN {X 0,Y 588.623,Z 440.838,A -85,B 0,C 180,E1 -1559.505,E2 -1559.505} C_VEL
LIN {X 0,Y 587.379,Z 434.696,A -85,B 0,C 180,E1 -1560.414,E2 -1560.414} C_VEL
LIN {X 0,Y 587.337,Z 434.572,A -85,B 0,C 180,E1 -1563.112,E2 -1563.112} C_VEL
LIN {X 0,Y 587.352,Z 434.571,A -85,B 0,C 180,E1 -1565.895,E2 -1565.895} C_VEL
LIN {X 0,Y 587.326,Z 434.565,A -85,B 0,C 180,E1 -1568.479,E2 -1568.479} C_VEL
LIN {X 0,Y 587.33,Z 434.572,A -85,B 0,C 180,E1 -1571.156,E2 -1571.156} C_VEL
LIN {X 0,Y 587.32,Z 434.574,A -85,B 0,C 180,E1 -1574.113,E2 -1574.113} C_VEL
LIN {X 0,Y 587.317,Z 434.57,A -85,B 0,C 180,E1 -1576.994,E2 -1576.994} C_VEL
LIN {X 0,Y 587.323,Z 434.578,A -85,B 0,C 180,E1 -1579.746,E2 -1579.746} C_VEL
LIN {X 0,Y 587.341,Z 434.569,A -85,B 0,C 180,E1 -1582.392,E2 -1582.392} C_VEL
LIN {X 0,Y 587.341,Z 434.564,A -85,B 0,C 180,E1 -1584.945,E2 -1584.945} C_VEL
LIN {X 0,Y 587.332,Z 434.57,A -85,B 0,C 180,E1 -1587.421,E2 -1587.421} C_VEL
LIN {X 0,Y 587.339,Z 434.575,A -85,B 0,C 180,E1 -1589.83,E2 -1589.83} C_VEL
LIN {X 0,Y 587.343,Z 434.57,A -85,B 0,C 180,E1 -1592.306,E2 -1592.306} C_VEL
LIN {X 0,Y 587.329,Z 434.572,A -85,B 0,C 180,E1 -1594.483,E2 -1594.483} C_VEL
LIN {X 0,Y 587.31,Z 434.57,A -85,B 0,C 180,E1 -1597.13,E2 -1597.13} C_VEL
LIN {X 0,Y 587.324,Z 434.568,A -85,B 0,C 180,E1 -1599.695,E2 -1599.695} C_VEL
LIN {X 0,Y 587.35,Z 434.569,A -85,B 0,C 180,E1 -1602.594,E2 -1602.594} C_VEL
LIN {X 0,Y 587.355,Z 434.567,A -85,B 0,C 180,E1 -1605.739,E2 -1605.739} C_VEL
LIN {X 0,Y 587.352,Z 434.568,A -85,B 0,C 180,E1 -1608.858,E2 -1608.858} C_VEL
LIN {X 0,Y 587.365,Z 434.564,A -85,B 0,C 180,E1 -1611.745,E2 -1611.745} C_VEL
LIN {X 0,Y 587.349,Z 434.574,A -85,B 0,C 180,E1 -1614.507,E2 -1614.507} C_VEL
LIN {X 0,Y 587.375,Z 434.562,A -85,B 0,C 180,E1 -1617.257,E2 -1617.257} C_VEL
LIN {X 0,Y 587.373,Z 434.566,A -85,B 0,C 180,E1 -1620,E2 -1620} C_VEL
LIN {X 0,Y 587.374,Z 434.57,A -85,B 0,C 180,E1 -1622.743,E2 -1622.743} C_VEL
LIN {X 0,Y 587.355,Z 434.564,A -85,B 0,C 180,E1 -1625.493,E2 -1625.493} C_VEL
LIN {X 0,Y 587.365,Z 434.568,A -85,B 0,C 180,E1 -1628.255,E2 -1628.255} C_VEL
LIN {X 0,Y 587.352,Z 434.567,A -85,B 0,C 180,E1 -1631.141,E2 -1631.141} C_VEL
LIN {X 0,Y 587.354,Z 434.568,A -85,B 0,C 180,E1 -1634.261,E2 -1634.261} C_VEL
LIN {X 0,Y 587.35,Z 434.567,A -85,B 0,C 180,E1 -1637.406,E2 -1637.406} C_VEL
LIN {X 0,Y 587.318,Z 434.572,A -85,B 0,C 180,E1 -1638.324,E2 -1638.324} C_VEL
LIN {X 0,Y 586.664,Z 434.66,A -85,B 0,C 180,E1 -1638.896,E2 -1638.896} C_VEL
LIN {X 0,Y 583.834,Z 435.015,A -85,B 0,C 180,E1 -1639.824,E2 -1639.824} C_VEL
LIN {X 0,Y 581.425,Z 435.313,A -85,B 0,C 180,E1 -1640.571,E2 -1640.571} C_VEL
LIN {X 0,Y 580.372,Z 435.441,A -85,B 0,C 180,E1 -1641.147,E2 -1641.147} C_VEL
LIN {X 0,Y 580.277,Z 435.45,A -85,B 0,C 180,E1 -1641.343,E2 -1641.343} C_VEL
LIN {X 0,Y 580.292,Z 435.446,A -85,B 0,C 180,E1 -1644.316,E2 -1644.316} C_VEL
LIN {X 0,Y 580.301,Z 435.444,A -85,B 0,C 180,E1 -1646.622,E2 -1646.622} C_VEL
LIN {X 0,Y 580.296,Z 435.45,A -85,B 0,C 180,E1 -1649.311,E2 -1649.311} C_VEL
LIN {X 0,Y 580.293,Z 435.444,A -85,B 0,C 180,E1 -1652.2,E2 -1652.2} C_VEL
LIN {X 0,Y 580.291,Z 435.444,A -85,B 0,C 180,E1 -1654.696,E2 -1654.696} C_VEL
LIN {X 0,Y 580.294,Z 435.453,A -85,B 0,C 180,E1 -1657.268,E2 -1657.268} C_VEL
LIN {X 0,Y 580.298,Z 435.445,A -85,B 0,C 180,E1 -1660.273,E2 -1660.273} C_VEL
LIN {X 0,Y 580.275,Z 435.45,A -85,B 0,C 180,E1 -1662.706,E2 -1662.706} C_VEL
LIN {X 0,Y 580.266,Z 435.453,A -85,B 0,C 180,E1 -1665.609,E2 -1665.609} C_VEL
LIN {X 0,Y 580.306,Z 435.444,A -85,B 0,C 180,E1 -1668.235,E2 -1668.235} C_VEL
LIN {X 0,Y 580.282,Z 435.451,A -85,B 0,C 180,E1 -1670.966,E2 -1670.966} C_VEL
LIN {X 0,Y 580.29,Z 435.452,A -85,B 0,C 180,E1 -1673.599,E2 -1673.599} C_VEL
LIN {X 0,Y 580.315,Z 435.444,A -85,B 0,C 180,E1 -1676.146,E2 -1676.146} C_VEL
LIN {X 0,Y 580.283,Z 435.447,A -85,B 0,C 180,E1 -1678.616,E2 -1678.616} C_VEL
LIN {X 0,Y 580.289,Z 435.449,A -85,B 0,C 180,E1 -1681.024,E2 -1681.024} C_VEL
LIN {X 0,Y 580.322,Z 435.451,A -85,B 0,C 180,E1 -1683.659,E2 -1683.659} C_VEL
LIN {X 0,Y 580.274,Z 435.448,A -85,B 0,C 180,E1 -1686.442,E2 -1686.442} C_VEL
LIN {X 0,Y 580.271,Z 435.455,A -85,B 0,C 180,E1 -1689.438,E2 -1689.438} C_VEL
LIN {X 0,Y 580.276,Z 435.457,A -85,B 0,C 180,E1 -1691.646,E2 -1691.646} C_VEL
LIN {X 0,Y 580.277,Z 435.457,A -85,B 0,C 180,E1 -1693.826,E2 -1693.826} C_VEL
LIN {X 0,Y 580.324,Z 435.448,A -85,B 0,C 180,E1 -1695.983,E2 -1695.983} C_VEL
LIN {X 0,Y 580.301,Z 435.445,A -85,B 0,C 180,E1 -1698.827,E2 -1698.827} C_VEL
LIN {X 0,Y 580.325,Z 435.448,A -85,B 0,C 180,E1 -1701.644,E2 -1701.644} C_VEL
LIN {X 0,Y 580.321,Z 435.445,A -85,B 0,C 180,E1 -1704.44,E2 -1704.44} C_VEL
LIN {X 0,Y 580.335,Z 435.441,A -85,B 0,C 180,E1 -1707.224,E2 -1707.224} C_VEL
LIN {X 0,Y 580.351,Z 435.449,A -85,B 0,C 180,E1 -1710,E2 -1710} C_VEL
LIN {X 0,Y 580.335,Z 435.441,A -85,B 0,C 180,E1 -1712.776,E2 -1712.776} C_VEL
LIN {X 0,Y 580.321,Z 435.444,A -85,B 0,C 180,E1 -1715.56,E2 -1715.56} C_VEL
LIN {X 0,Y 580.325,Z 435.448,A -85,B 0,C 180,E1 -1718.356,E2 -1718.356} C_VEL
LIN {X 0,Y 580.296,Z 435.445,A -85,B 0,C 180,E1 -1721.191,E2 -1721.191} C_VEL
LIN {X 0,Y 580.324,Z 435.448,A -85,B 0,C 180,E1 -1724.017,E2 -1724.017} C_VEL
LIN {X 0,Y 580.308,Z 435.445,A -85,B 0,C 180,E1 -1726.914,E2 -1726.914} C_VEL
LIN {X 0,Y 580.301,Z 435.447,A -85,B 0,C 180,E1 -1729.822,E2 -1729.822} C_VEL
LIN {X 0,Y 580.29,Z 435.45,A -85,B 0,C 180,E1 -1732.802,E2 -1732.802} C_VEL
LIN {X 0,Y 580.303,Z 435.445,A -85,B 0,C 180,E1 -1735.079,E2 -1735.079} C_VEL
LIN {X 0,Y 580.315,Z 435.444,A -85,B 0,C 180,E1 -1737.863,E2 -1737.863} C_VEL
LIN {X 0,Y 580.285,Z 435.454,A -85,B 0,C 180,E1 -1740.696,E2 -1740.696} C_VEL
LIN {X 0,Y 580.3,Z 435.445,A -85,B 0,C 180,E1 -1743.317,E2 -1743.317} C_VEL
LIN {X 0,Y 580.32,Z 435.442,A -85,B 0,C 180,E1 -1745.767,E2 -1745.767} C_VEL
LIN {X 0,Y 580.281,Z 435.45,A -85,B 0,C 180,E1 -1748.146,E2 -1748.146} C_VEL
LIN {X 0,Y 580.292,Z 435.453,A -85,B 0,C 180,E1 -1750.843,E2 -1750.843} C_VEL
LIN {X 0,Y 580.279,Z 435.447,A -85,B 0,C 180,E1 -1753.657,E2 -1753.657} C_VEL
LIN {X 0,Y 580.278,Z 435.455,A -85,B 0,C 180,E1 -1756.608,E2 -1756.608} C_VEL
LIN {X 0,Y 580.311,Z 435.448,A -85,B 0,C 180,E1 -1759.158,E2 -1759.158} C_VEL
LIN {X 0,Y 580.284,Z 435.446,A -85,B 0,C 180,E1 -1761.926,E2 -1761.926} C_VEL
LIN {X 0,Y 580.297,Z 435.447,A -85,B 0,C 180,E1 -1764.456,E2 -1764.456} C_VEL
LIN {X 0,Y 580.282,Z 435.452,A -85,B 0,C 180,E1 -1766.975,E2 -1766.975} C_VEL
LIN {X 0,Y 580.301,Z 435.448,A -85,B 0,C 180,E1 -1769.426,E2 -1769.426} C_VEL
LIN {X 0,Y 580.31,Z 435.44,A -85,B 0,C 180,E1 -1772.137,E2 -1772.137} C_VEL
LIN {X 0,Y 580.299,Z 435.447,A -85,B 0,C 180,E1 -1774.92,E2 -1774.92} C_VEL
LIN {X 0,Y 580.264,Z 435.449,A -85,B 0,C 180,E1 -1777.947,E2 -1777.947} C_VEL
LIN {X 0,Y 580.308,Z 435.448,A -85,B 0,C 180,E1 -1780.914,E2 -1780.914} C_VEL
LIN {X 0,Y 580.272,Z 435.447,A -85,B 0,C 180,E1 -1783.826,E2 -1783.826} C_VEL
LIN {X 0,Y 580.316,Z 435.443,A -85,B 0,C 180,E1 -1785.983,E2 -1785.983} C_VEL
LIN {X 0,Y 580.321,Z 435.443,A -85,B 0,C 180,E1 -1788.827,E2 -1788.827} C_VEL
LIN {X 0,Y 580.328,Z 435.446,A -85,B 0,C 180,E1 -1791.644,E2 -1791.644} C_VEL
LIN {X 0,Y 580.322,Z 435.44,A -85,B 0,C 180,E1 -1794.44,E2 -1794.44} C_VEL
LIN {X 0,Y 580.339,Z 435.446,A -85,B 0,C 180,E1 -1797.224,E2 -1797.224} C_VEL
LIN {X 0,Y 580.342,Z 435.442,A -85,B 0,C 180,E1 -1800,E2 -1800} C_VEL
LIN {X 0,Y 580.34,Z 435.439,A -85,B 0,C 180,E1 -1802.777,E2 -1802.777} C_VEL
LIN {X 0,Y 580.315,Z 435.452,A -85,B 0,C 180,E1 -1805.56,E2 -1805.56} C_VEL
LIN {X 0,Y 580.328,Z 435.439,A -85,B 0,C 180,E1 -1808.356,E2 -1808.356} C_VEL
LIN {X 0,Y 580.323,Z 435.444,A -85,B 0,C 180,E1 -1811.209,E2 -1811.209} C_VEL
LIN {X 0,Y 580.305,Z 435.445,A -85,B 0,C 180,E1 -1814.339,E2 -1814.339} C_VEL
LIN {X 0,Y 580.302,Z 435.443,A -85,B 0,C 180,E1 -1816.914,E2 -1816.914} C_VEL
LIN {X 0,Y 580.298,Z 435.447,A -85,B 0,C 180,E1 -1819.823,E2 -1819.823} C_VEL
LIN {X 0,Y 580.265,Z 435.455,A -85,B 0,C 180,E1 -1822.053,E2 -1822.053} C_VEL
LIN {X 0,Y 580.3,Z 435.444,A -85,B 0,C 180,E1 -1825.08,E2 -1825.08} C_VEL
LIN {X 0,Y 580.311,Z 435.448,A -85,B 0,C 180,E1 -1827.864,E2 -1827.864} C_VEL
LIN {X 0,Y 580.292,Z 435.446,A -85,B 0,C 180,E1 -1830.698,E2 -1830.698} C_VEL
LIN {X 0,Y 580.296,Z 435.445,A -85,B 0,C 180,E1 -1833.317,E2 -1833.317} C_VEL
LIN {X 0,Y 580.317,Z 435.443,A -85,B 0,C 180,E1 -1835.768,E2 -1835.768} C_VEL
LIN {X 0,Y 580.284,Z 435.456,A -85,B 0,C 180,E1 -1838.147,E2 -1838.147} C_VEL
LIN {X 0,Y 580.299,Z 435.445,A -85,B 0,C 180,E1 -1840.843,E2 -1840.843} C_VEL
LIN {X 0,Y 580.282,Z 435.448,A -85,B 0,C 180,E1 -1843.657,E2 -1843.657} C_VEL
LIN {X 0,Y 580.27,Z 435.452,A -85,B 0,C 180,E1 -1846.61,E2 -1846.61} C_VEL
LIN {X 0,Y 580.294,Z 435.446,A -85,B 0,C 180,E1 -1849.157,E2 -1849.157} C_VEL
LIN {X 0,Y 580.284,Z 435.445,A -85,B 0,C 180,E1 -1851.928,E2 -1851.928} C_VEL
LIN {X 0,Y 580.303,Z 435.453,A -85,B 0,C 180,E1 -1854.457,E2 -1854.457} C_VEL
LIN {X 0,Y 580.289,Z 435.449,A -85,B 0,C 180,E1 -1856.976,E2 -1856.976} C_VEL
LIN {X 0,Y 580.32,Z 435.621,A -85,B 0,C 180,E1 -1859.299,E2 -1859.299} C_VEL
LIN {X 0,Y 581.881,Z 442.331,A -85,B 0,C 180,E1 -1860.318,E2 -1860.318} C_VEL
LIN {X 0,Y 581.561,Z 464.922,A -85,B 0,C 180,E1 -1863.267,E2 -1863.267} C_VEL
LIN {X 0,Y 581.351,Z 484.296,A -85,B 0,C 180,E1 -1865.71,E2 -1865.71} C_VEL
LIN {X 0,Y 582.914,Z 490.746,A -85,B 0,C 180,E1 -1865.887,E2 -1865.887} C_VEL
LIN {X 0,Y 582.349,Z 689.076,A -85,B 0,C 180,E1 -1868.463,E2 -1868.463} C_VEL
LIN {X 0,Y 582.232,Z 706.479,A -85,B 0,C 180,E1 -1868.77,E2 -1868.77} C_VEL
LIN {X 0,Y 582.071,Z 722.111,A -85,B 0,C 180,E1 -1869.181,E2 -1869.181} C_VEL
LIN {X 0,Y 581.882,Z 738.065,A -85,B 0,C 180,E1 -1869.728,E2 -1869.728} C_VEL
LIN {X 0,Y 581.684,Z 754.641,A -85,B 0,C 180,E1 -1870.459,E2 -1870.459} C_VEL
LIN {X 0,Y 581.396,Z 770.368,A -85,B 0,C 180,E1 -1871.317,E2 -1871.317} C_VEL
LIN {X 0,Y 581.154,Z 784.185,A -85,B 0,C 180,E1 -1872.221,E2 -1872.221} C_VEL
LIN {X 0,Y 580.944,Z 798.264,A -85,B 0,C 180,E1 -1873.303,E2 -1873.303} C_VEL
LIN {X 0,Y 580.763,Z 810.278,A -85,B 0,C 180,E1 -1874.38,E2 -1874.38} C_VEL
LIN {X 0,Y 580.564,Z 821.646,A -85,B 0,C 180,E1 -1875.566,E2 -1875.566} C_VEL
LIN {X 0,Y 580.431,Z 832.445,A -85,B 0,C 180,E1 -1876.878,E2 -1876.878} C_VEL
LIN {X 0,Y 580.299,Z 842.475,A -85,B 0,C 180,E1 -1878.296,E2 -1878.296} C_VEL
LIN {X 0,Y 580.228,Z 849.918,A -85,B 0,C 180,E1 -1879.532,E2 -1879.532} C_VEL
LIN {X 0,Y 580.146,Z 857.134,A -85,B 0,C 180,E1 -1880.939,E2 -1880.939} C_VEL
LIN {X 0,Y 580.116,Z 863.151,A -85,B 0,C 180,E1 -1882.342,E2 -1882.342} C_VEL
LIN {X 0,Y 580.074,Z 867.958,A -85,B 0,C 180,E1 -1883.74,E2 -1883.74} C_VEL
LIN {X 0,Y 580.03,Z 871.797,A -85,B 0,C 180,E1 -1885.135,E2 -1885.135} C_VEL
LIN {X 0,Y 580.104,Z 874.564,A -85,B 0,C 180,E1 -1886.527,E2 -1886.527} C_VEL
LIN {X 0,Y 580.033,Z 876.439,A -85,B 0,C 180,E1 -1887.917,E2 -1887.917} C_VEL
LIN {X 0,Y 580.035,Z 877.35,A -85,B 0,C 180,E1 -1889.306,E2 -1889.306} C_VEL
LIN {X 0,Y 580.035,Z 877.35,A -85,B 0,C 180,E1 -1890.694,E2 -1890.694} C_VEL
LIN {X 0,Y 580.033,Z 876.439,A -85,B 0,C 180,E1 -1892.083,E2 -1892.083} C_VEL
LIN {X 0,Y 580.104,Z 874.564,A -85,B 0,C 180,E1 -1893.473,E2 -1893.473} C_VEL
LIN {X 0,Y 580.03,Z 871.797,A -85,B 0,C 180,E1 -1894.865,E2 -1894.865} C_VEL
LIN {X 0,Y 580.074,Z 867.958,A -85,B 0,C 180,E1 -1896.26,E2 -1896.26} C_VEL
LIN {X 0,Y 580.116,Z 863.151,A -85,B 0,C 180,E1 -1897.658,E2 -1897.658} C_VEL
LIN {X 0,Y 580.146,Z 857.134,A -85,B 0,C 180,E1 -1899.061,E2 -1899.061} C_VEL
LIN {X 0,Y 580.202,Z 848.905,A -85,B 0,C 180,E1 -1900.645,E2 -1900.645} C_VEL
LIN {X 0,Y 580.319,Z 840.135,A -85,B 0,C 180,E1 -1902.058,E2 -1902.058} C_VEL
LIN {X 0,Y 580.465,Z 829.715,A -85,B 0,C 180,E1 -1903.478,E2 -1903.478} C_VEL
LIN {X 0,Y 580.639,Z 817.357,A -85,B 0,C 180,E1 -1904.904,E2 -1904.904} C_VEL
LIN {X 0,Y 580.822,Z 804.477,A -85,B 0,C 180,E1 -1906.158,E2 -1906.158} C_VEL
LIN {X 0,Y 581.025,Z 792.718,A -85,B 0,C 180,E1 -1907.144,E2 -1907.144} C_VEL
LIN {X 0,Y 581.274,Z 778.998,A -85,B 0,C 180,E1 -1908.139,E2 -1908.139} C_VEL
LIN {X 0,Y 581.526,Z 764.135,A -85,B 0,C 180,E1 -1909.044,E2 -1909.044} C_VEL
LIN {X 0,Y 581.733,Z 747.775,A -85,B 0,C 180,E1 -1909.863,E2 -1909.863} C_VEL
LIN {X 0,Y 581.961,Z 731.888,A -85,B 0,C 180,E1 -1910.5,E2 -1910.5} C_VEL
LIN {X 0,Y 582.173,Z 714.998,A -85,B 0,C 180,E1 -1911.024,E2 -1911.024} C_VEL
LIN {X 0,Y 582.307,Z 697.83,A -85,B 0,C 180,E1 -1911.401,E2 -1911.401} C_VEL
LIN {X 0,Y 582.472,Z 652.36,A -85,B 0,C 180,E1 -1912.011,E2 -1912.011} C_VEL
LIN {X 0,Y 582.907,Z 490.768,A -85,B 0,C 180,E1 -1914.113,E2 -1914.113} C_VEL
LIN {X 0,Y 581.339,Z 484.293,A -85,B 0,C 180,E1 -1914.29,E2 -1914.29} C_VEL
LIN {X 0,Y 581.562,Z 464.922,A -85,B 0,C 180,E1 -1916.733,E2 -1916.733} C_VEL
LIN {X 0,Y 581.912,Z 443.003,A -85,B 0,C 180,E1 -1919.591,E2 -1919.591} C_VEL
LIN {X 0,Y 580.857,Z 437.844,A -85,B 0,C 180,E1 -1920.34,E2 -1920.34} C_VEL
LIN {X 0,Y 580.315,Z 435.496,A -85,B 0,C 180,E1 -1920.741,E2 -1920.741} C_VEL
LIN {X 0,Y 580.316,Z 435.443,A -85,B 0,C 180,E1 -1923.854,E2 -1923.854} C_VEL
LIN {X 0,Y 580.291,Z 435.446,A -85,B 0,C 180,E1 -1926.401,E2 -1926.401} C_VEL
LIN {X 0,Y 580.302,Z 435.443,A -85,B 0,C 180,E1 -1929.186,E2 -1929.186} C_VEL
LIN {X 0,Y 580.283,Z 435.454,A -85,B 0,C 180,E1 -1931.767,E2 -1931.767} C_VEL
LIN {X 0,Y 580.26,Z 435.449,A -85,B 0,C 180,E1 -1934.625,E2 -1934.625} C_VEL
LIN {X 0,Y 580.276,Z 435.45,A -85,B 0,C 180,E1 -1937.294,E2 -1937.294} C_VEL
LIN {X 0,Y 580.292,Z 435.45,A -85,B 0,C 180,E1 -1940.067,E2 -1940.067} C_VEL
LIN {X 0,Y 580.295,Z 435.445,A -85,B 0,C 180,E1 -1943.064,E2 -1943.064} C_VEL
LIN {X 0,Y 580.296,Z 435.444,A -85,B 0,C 180,E1 -1945.44,E2 -1945.44} C_VEL
LIN {X 0,Y 580.301,Z 435.455,A -85,B 0,C 180,E1 -1947.967,E2 -1947.967} C_VEL
LIN {X 0,Y 580.297,Z 435.441,A -85,B 0,C 180,E1 -1950.689,E2 -1950.689} C_VEL
LIN {X 0,Y 580.319,Z 435.443,A -85,B 0,C 180,E1 -1953.658,E2 -1953.658} C_VEL
LIN {X 0,Y 580.273,Z 435.451,A -85,B 0,C 180,E1 -1956.442,E2 -1956.442} C_VEL
LIN {X 0,Y 580.273,Z 435.443,A -85,B 0,C 180,E1 -1959.437,E2 -1959.437} C_VEL
LIN {X 0,Y 580.273,Z 435.445,A -85,B 0,C 180,E1 -1961.645,E2 -1961.645} C_VEL
LIN {X 0,Y 580.272,Z 435.451,A -85,B 0,C 180,E1 -1963.825,E2 -1963.825} C_VEL
LIN {X 0,Y 580.316,Z 435.447,A -85,B 0,C 180,E1 -1965.983,E2 -1965.983} C_VEL
LIN {X 0,Y 580.322,Z 435.444,A -85,B 0,C 180,E1 -1968.827,E2 -1968.827} C_VEL
LIN {X 0,Y 580.328,Z 435.439,A -85,B 0,C 180,E1 -1971.644,E2 -1971.644} C_VEL
LIN {X 0,Y 580.315,Z 435.452,A -85,B 0,C 180,E1 -1974.44,E2 -1974.44} C_VEL
LIN {X 0,Y 580.34,Z 435.439,A -85,B 0,C 180,E1 -1977.223,E2 -1977.223} C_VEL
LIN {X 0,Y 580.342,Z 435.442,A -85,B 0,C 180,E1 -1980,E2 -1980} C_VEL
LIN {X 0,Y 580.339,Z 435.445,A -85,B 0,C 180,E1 -1982.776,E2 -1982.776} C_VEL
LIN {X 0,Y 580.322,Z 435.44,A -85,B 0,C 180,E1 -1985.56,E2 -1985.56} C_VEL
LIN {X 0,Y 580.328,Z 435.446,A -85,B 0,C 180,E1 -1988.356,E2 -1988.356} C_VEL
LIN {X 0,Y 580.323,Z 435.442,A -85,B 0,C 180,E1 -1991.208,E2 -1991.208} C_VEL
LIN {X 0,Y 580.304,Z 435.448,A -85,B 0,C 180,E1 -1994.339,E2 -1994.339} C_VEL
LIN {X 0,Y 580.302,Z 435.452,A -85,B 0,C 180,E1 -1996.914,E2 -1996.914} C_VEL
LIN {X 0,Y 580.297,Z 435.443,A -85,B 0,C 180,E1 -1999.822,E2 -1999.822} C_VEL
LIN {X 0,Y 580.277,Z 435.45,A -85,B 0,C 180,E1 -2001.343,E2 -2001.343} C_VEL
LIN {X 0,Y 579.579,Z 435.537,A -85,B 0,C 180,E1 -2001.922,E2 -2001.922} C_VEL
LIN {X 0,Y 576.702,Z 435.903,A -85,B 0,C 180,E1 -2002.862,E2 -2002.862} C_VEL
LIN {X 0,Y 574.307,Z 436.195,A -85,B 0,C 180,E1 -2003.618,E2 -2003.618} C_VEL
LIN {X 0,Y 573.308,Z 436.316,A -85,B 0,C 180,E1 -2004.202,E2 -2004.202} C_VEL
LIN {X 0,Y 573.242,Z 436.325,A -85,B 0,C 180,E1 -2004.399,E2 -2004.399} C_VEL
LIN {X 0,Y 573.258,Z 436.323,A -85,B 0,C 180,E1 -2006.975,E2 -2006.975} C_VEL
LIN {X 0,Y 573.244,Z 436.326,A -85,B 0,C 180,E1 -2009.49,E2 -2009.49} C_VEL
LIN {X 0,Y 573.246,Z 436.322,A -85,B 0,C 180,E1 -2012.229,E2 -2012.229} C_VEL
LIN {X 0,Y 573.241,Z 436.322,A -85,B 0,C 180,E1 -2014.774,E2 -2014.774} C_VEL
LIN {X 0,Y 573.247,Z 436.333,A -85,B 0,C 180,E1 -2017.167,E2 -2017.167} C_VEL
LIN {X 0,Y 573.242,Z 436.327,A -85,B 0,C 180,E1 -2019.607,E2 -2019.607} C_VEL
LIN {X 0,Y 573.233,Z 436.325,A -85,B 0,C 180,E1 -2022.4,E2 -2022.4} C_VEL
LIN {X 0,Y 573.219,Z 436.329,A -85,B 0,C 180,E1 -2024.676,E2 -2024.676} C_VEL
LIN {X 0,Y 573.235,Z 436.334,A -85,B 0,C 180,E1 -2027.358,E2 -2027.358} C_VEL
LIN {X 0,Y 573.241,Z 436.324,A -85,B 0,C 180,E1 -2030.394,E2 -2030.394} C_VEL
LIN {X 0,Y 573.249,Z 436.329,A -85,B 0,C 180,E1 -2033.078,E2 -2033.078} C_VEL
LIN {X 0,Y 573.269,Z 436.327,A -85,B 0,C 180,E1 -2035.672,E2 -2035.672} C_VEL
LIN {X 0,Y 573.244,Z 436.324,A -85,B 0,C 180,E1 -2038.186,E2 -2038.186} C_VEL
LIN {X 0,Y 573.26,Z 436.322,A -85,B 0,C 180,E1 -2040.635,E2 -2040.635} C_VEL
LIN {X 0,Y 573.264,Z 436.33,A -85,B 0,C 180,E1 -2043.501,E2 -2043.501} C_VEL
LIN {X 0,Y 573.227,Z 436.328,A -85,B 0,C 180,E1 -2046.135,E2 -2046.135} C_VEL
LIN {X 0,Y 573.247,Z 436.326,A -85,B 0,C 180,E1 -2049.174,E2 -2049.174} C_VEL
LIN {X 0,Y 573.233,Z 436.331,A -85,B 0,C 180,E1 -2051.412,E2 -2051.412} C_VEL
LIN {X 0,Y 573.254,Z 436.331,A -85,B 0,C 180,E1 -2053.622,E2 -2053.622} C_VEL
LIN {X 0,Y 573.234,Z 436.326,A -85,B 0,C 180,E1 -2056.53,E2 -2056.53} C_VEL
LIN {X 0,Y 573.259,Z 436.322,A -85,B 0,C 180,E1 -2058.745,E2 -2058.745} C_VEL
LIN {X 0,Y 573.281,Z 436.324,A -85,B 0,C 180,E1 -2061.541,E2 -2061.541} C_VEL
LIN {X 0,Y 573.288,Z 436.322,A -85,B 0,C 180,E1 -2064.372,E2 -2064.372} C_VEL
LIN {X 0,Y 573.31,Z 436.325,A -85,B 0,C 180,E1 -2067.892,E2 -2067.892} C_VEL
LIN {X 0,Y 573.326,Z 436.315,A -85,B 0,C 180,E1 -2070.702,E2 -2070.702} C_VEL
LIN {X 0,Y 573.301,Z 436.317,A -85,B 0,C 180,E1 -2072.811,E2 -2072.811} C_VEL
LIN {X 0,Y 573.288,Z 436.322,A -85,B 0,C 180,E1 -2075.628,E2 -2075.628} C_VEL
LIN {X 0,Y 573.281,Z 436.324,A -85,B 0,C 180,E1 -2078.459,E2 -2078.459} C_VEL
LIN {X 0,Y 573.268,Z 436.321,A -85,B 0,C 180,E1 -2081.312,E2 -2081.312} C_VEL
LIN {X 0,Y 573.27,Z 436.33,A -85,B 0,C 180,E1 -2084.193,E2 -2084.193} C_VEL
LIN {X 0,Y 573.256,Z 436.322,A -85,B 0,C 180,E1 -2087.111,E2 -2087.111} C_VEL
LIN {X 0,Y 573.249,Z 436.329,A -85,B 0,C 180,E1 -2090.076,E2 -2090.076} C_VEL
LIN {X 0,Y 573.229,Z 436.327,A -85,B 0,C 180,E1 -2093.099,E2 -2093.099} C_VEL
LIN {X 0,Y 573.25,Z 436.323,A -85,B 0,C 180,E1 -2095.41,E2 -2095.41} C_VEL
LIN {X 0,Y 573.259,Z 436.325,A -85,B 0,C 180,E1 -2098.031,E2 -2098.031} C_VEL
LIN {X 0,Y 573.232,Z 436.33,A -85,B 0,C 180,E1 -2100.883,E2 -2100.883} C_VEL
LIN {X 0,Y 573.282,Z 436.319,A -85,B 0,C 180,E1 -2103.528,E2 -2103.528} C_VEL
LIN {X 0,Y 573.255,Z 436.324,A -85,B 0,C 180,E1 -2106.048,E2 -2106.048} C_VEL
LIN {X 0,Y 573.241,Z 436.334,A -85,B 0,C 180,E1 -2108.701,E2 -2108.701} C_VEL
LIN {X 0,Y 573.245,Z 436.323,A -85,B 0,C 180,E1 -2111.595,E2 -2111.595} C_VEL
LIN {X 0,Y 573.231,Z 436.329,A -85,B 0,C 180,E1 -2114.333,E2 -2114.333} C_VEL
LIN {X 0,Y 573.236,Z 436.327,A -85,B 0,C 180,E1 -2117.358,E2 -2117.358} C_VEL
LIN {X 0,Y 573.265,Z 436.322,A -85,B 0,C 180,E1 -2119.477,E2 -2119.477} C_VEL
LIN {X 0,Y 573.229,Z 436.326,A -85,B 0,C 180,E1 -2122.192,E2 -2122.192} C_VEL
LIN {X 0,Y 573.259,Z 436.328,A -85,B 0,C 180,E1 -2124.816,E2 -2124.816} C_VEL
LIN {X 0,Y 573.247,Z 436.326,A -85,B 0,C 180,E1 -2127.355,E2 -2127.355} C_VEL
LIN {X 0,Y 573.247,Z 436.323,A -85,B 0,C 180,E1 -2129.824,E2 -2129.824} C_VEL
LIN {X 0,Y 573.279,Z 436.315,A -85,B 0,C 180,E1 -2132.235,E2 -2132.235} C_VEL
LIN {X 0,Y 573.259,Z 436.327,A -85,B 0,C 180,E1 -2135.121,E2 -2135.121} C_VEL
LIN {X 0,Y 573.228,Z 436.328,A -85,B 0,C 180,E1 -2137.662,E2 -2137.662} C_VEL
LIN {X 0,Y 573.247,Z 436.322,A -85,B 0,C 180,E1 -2139.923,E2 -2139.923} C_VEL
LIN {X 0,Y 573.251,Z 436.329,A -85,B 0,C 180,E1 -2142.989,E2 -2142.989} C_VEL
LIN {X 0,Y 573.263,Z 436.323,A -85,B 0,C 180,E1 -2145.807,E2 -2145.807} C_VEL
LIN {X 0,Y 573.273,Z 436.319,A -85,B 0,C 180,E1 -2148.734,E2 -2148.734} C_VEL
LIN {X 0,Y 573.299,Z 436.323,A -85,B 0,C 180,E1 -2151.541,E2 -2151.541} C_VEL
LIN {X 0,Y 573.289,Z 436.316,A -85,B 0,C 180,E1 -2154.372,E2 -2154.372} C_VEL
LIN {X 0,Y 573.299,Z 436.317,A -85,B 0,C 180,E1 -2157.893,E2 -2157.893} C_VEL
LIN {X 0,Y 573.328,Z 436.313,A -85,B 0,C 180,E1 -2160.703,E2 -2160.703} C_VEL
LIN {X 0,Y 573.232,Z 436.333,A -85,B 0,C 180,E1 -2163.515,E2 -2163.515} C_VEL
LIN {X 0,Y 573.282,Z 436.329,A -85,B 0,C 180,E1 -2165.628,E2 -2165.628} C_VEL
LIN {X 0,Y 573.299,Z 436.314,A -85,B 0,C 180,E1 -2168.459,E2 -2168.459} C_VEL
LIN {X 0,Y 573.289,Z 436.321,A -85,B 0,C 180,E1 -2171.312,E2 -2171.312} C_VEL
LIN {X 0,Y 573.271,Z 436.32,A -85,B 0,C 180,E1 -2174.425,E2 -2174.425} C_VEL
LIN {X 0,Y 573.25,Z 436.323,A -85,B 0,C 180,E1 -2177.112,E2 -2177.112} C_VEL
LIN {X 0,Y 573.247,Z 436.323,A -85,B 0,C 180,E1 -2180.077,E2 -2180.077} C_VEL
LIN {X 0,Y 573.229,Z 436.327,A -85,B 0,C 180,E1 -2182.338,E2 -2182.338} C_VEL
LIN {X 0,Y 573.248,Z 436.325,A -85,B 0,C 180,E1 -2185.41,E2 -2185.41} C_VEL
LIN {X 0,Y 573.255,Z 436.323,A -85,B 0,C 180,E1 -2188.032,E2 -2188.032} C_VEL
LIN {X 0,Y 573.236,Z 436.324,A -85,B 0,C 180,E1 -2190.885,E2 -2190.885} C_VEL
LIN {X 0,Y 573.254,Z 436.324,A -85,B 0,C 180,E1 -2193.525,E2 -2193.525} C_VEL
LIN {X 0,Y 573.253,Z 436.327,A -85,B 0,C 180,E1 -2196.049,E2 -2196.049} C_VEL
LIN {X 0,Y 573.244,Z 436.324,A -85,B 0,C 180,E1 -2198.701,E2 -2198.701} C_VEL
LIN {X 0,Y 573.248,Z 436.324,A -85,B 0,C 180,E1 -2201.596,E2 -2201.596} C_VEL
LIN {X 0,Y 573.233,Z 436.332,A -85,B 0,C 180,E1 -2204.334,E2 -2204.334} C_VEL
LIN {X 0,Y 573.234,Z 436.323,A -85,B 0,C 180,E1 -2207.359,E2 -2207.359} C_VEL
LIN {X 0,Y 573.242,Z 436.328,A -85,B 0,C 180,E1 -2210.394,E2 -2210.394} C_VEL
LIN {X 0,Y 573.251,Z 436.324,A -85,B 0,C 180,E1 -2213.078,E2 -2213.078} C_VEL
LIN {X 0,Y 573.27,Z 436.319,A -85,B 0,C 180,E1 -2215.672,E2 -2215.672} C_VEL
LIN {X 0,Y 573.242,Z 436.321,A -85,B 0,C 180,E1 -2218.598,E2 -2218.598} C_VEL
LIN {X 0,Y 573.301,Z 436.539,A -85,B 0,C 180,E1 -2219.012,E2 -2219.012} C_VEL
LIN {X 0,Y 575.151,Z 444.131,A -85,B 0,C 180,E1 -2220.178,E2 -2220.178} C_VEL
LIN {X 0,Y 574.796,Z 466.267,A -85,B 0,C 180,E1 -2223.103,E2 -2223.103} C_VEL
LIN {X 0,Y 574.508,Z 484.118,A -85,B 0,C 180,E1 -2225.388,E2 -2225.388} C_VEL
LIN {X 0,Y 575.446,Z 488.164,A -85,B 0,C 180,E1 -2225.519,E2 -2225.519} C_VEL
LIN {X 0,Y 576.474,Z 493.071,A -85,B 0,C 180,E1 -2225.631,E2 -2225.631} C_VEL
LIN {X 0,Y 575.746,Z 695.228,A -85,B 0,C 180,E1 -2228.301,E2 -2228.301} C_VEL
LIN {X 0,Y 575.539,Z 711.357,A -85,B 0,C 180,E1 -2228.628,E2 -2228.628} C_VEL
LIN {X 0,Y 575.317,Z 729.308,A -85,B 0,C 180,E1 -2229.159,E2 -2229.159} C_VEL
LIN {X 0,Y 575.049,Z 745.716,A -85,B 0,C 180,E1 -2229.803,E2 -2229.803} C_VEL
LIN {X 0,Y 574.815,Z 760.009,A -85,B 0,C 180,E1 -2230.502,E2 -2230.502} C_VEL
LIN {X 0,Y 574.514,Z 774.773,A -85,B 0,C 180,E1 -2231.363,E2 -2231.363} C_VEL
LIN {X 0,Y 574.217,Z 790.097,A -85,B 0,C 180,E1 -2232.439,E2 -2232.439} C_VEL
LIN {X 0,Y 573.914,Z 803.468,A -85,B 0,C 180,E1 -2233.55,E2 -2233.55} C_VEL
LIN {X 0,Y 573.701,Z 815.597,A -85,B 0,C 180,E1 -2234.73,E2 -2234.73} C_VEL
LIN {X 0,Y 573.541,Z 826.801,A -85,B 0,C 180,E1 -2235.995,E2 -2235.995} C_VEL
LIN {X 0,Y 573.342,Z 837.675,A -85,B 0,C 180,E1 -2237.433,E2 -2237.433} C_VEL
LIN {X 0,Y 573.232,Z 846.24,A -85,B 0,C 180,E1 -2238.76,E2 -2238.76} C_VEL
LIN {X 0,Y 573.147,Z 853.666,A -85,B 0,C 180,E1 -2240.115,E2 -2240.115} C_VEL
LIN {X 0,Y 573.078,Z 860.291,A -85,B 0,C 180,E1 -2241.538,E2 -2241.538} C_VEL
LIN {X 0,Y 573.044,Z 865.667,A -85,B 0,C 180,E1 -2242.955,E2 -2242.955} C_VEL
LIN {X 0,Y 573.037,Z 870.026,A -85,B 0,C 180,E1 -2244.369,E2 -2244.369} C_VEL
LIN {X 0,Y 573.003,Z 873.295,A -85,B 0,C 180,E1 -2245.78,E2 -2245.78} C_VEL
LIN {X 0,Y 572.95,Z 875.655,A -85,B 0,C 180,E1 -2247.188,E2 -2247.188} C_VEL
LIN {X 0,Y 572.939,Z 877.004,A -85,B 0,C 180,E1 -2248.594,E2 -2248.594} C_VEL
LIN {X 0,Y 572.933,Z 877.5,A -85,B 0,C 180,E1 -2250,E2 -2250} C_VEL
LIN {X 0,Y 572.939,Z 877.004,A -85,B 0,C 180,E1 -2251.406,E2 -2251.406} C_VEL
LIN {X 0,Y 572.95,Z 875.655,A -85,B 0,C 180,E1 -2252.812,E2 -2252.812} C_VEL
LIN {X 0,Y 573.003,Z 873.295,A -85,B 0,C 180,E1 -2254.22,E2 -2254.22} C_VEL
LIN {X 0,Y 573.037,Z 870.026,A -85,B 0,C 180,E1 -2255.631,E2 -2255.631} C_VEL
LIN {X 0,Y 573.044,Z 865.667,A -85,B 0,C 180,E1 -2257.045,E2 -2257.045} C_VEL
LIN {X 0,Y 573.078,Z 860.291,A -85,B 0,C 180,E1 -2258.462,E2 -2258.462} C_VEL
LIN {X 0,Y 573.147,Z 853.666,A -85,B 0,C 180,E1 -2259.885,E2 -2259.885} C_VEL
LIN {X 0,Y 573.245,Z 844.722,A -85,B 0,C 180,E1 -2261.491,E2 -2261.491} C_VEL
LIN {X 0,Y 573.382,Z 835.165,A -85,B 0,C 180,E1 -2262.926,E2 -2262.926} C_VEL
LIN {X 0,Y 573.563,Z 823.513,A -85,B 0,C 180,E1 -2264.398,E2 -2264.398} C_VEL
LIN {X 0,Y 573.78,Z 812.053,A -85,B 0,C 180,E1 -2265.632,E2 -2265.632} C_VEL
LIN {X 0,Y 574.028,Z 798.269,A -85,B 0,C 180,E1 -2266.904,E2 -2266.904} C_VEL
LIN {X 0,Y 574.336,Z 784.185,A -85,B 0,C 180,E1 -2267.997,E2 -2267.997} C_VEL
LIN {X 0,Y 574.586,Z 770.357,A -85,B 0,C 180,E1 -2268.913,E2 -2268.913} C_VEL
LIN {X 0,Y 574.909,Z 754.552,A -85,B 0,C 180,E1 -2269.785,E2 -2269.785} C_VEL
LIN {X 0,Y 575.186,Z 738.073,A -85,B 0,C 180,E1 -2270.519,E2 -2270.519} C_VEL
LIN {X 0,Y 575.426,Z 722.105,A -85,B 0,C 180,E1 -2271.071,E2 -2271.071} C_VEL
LIN {X 0,Y 575.612,Z 705.76,A -85,B 0,C 180,E1 -2271.503,E2 -2271.503} C_VEL
LIN {X 0,Y 575.751,Z 688.13,A -85,B 0,C 180,E1 -2271.81,E2 -2271.81} C_VEL
LIN {X 0,Y 576.435,Z 498.55,A -85,B 0,C 180,E1 -2274.297,E2 -2274.297} C_VEL
LIN {X 0,Y 576.301,Z 491.545,A -85,B 0,C 180,E1 -2274.397,E2 -2274.397} C_VEL
LIN {X 0,Y 574.539,Z 484.376,A -85,B 0,C 180,E1 -2274.593,E2 -2274.593} C_VEL
LIN {X 0,Y 574.633,Z 475.243,A -85,B 0,C 180,E1 -2275.732,E2 -2275.732} C_VEL
LIN {X 0,Y 574.983,Z 454.299,A -85,B 0,C 180,E1 -2278.469,E2 -2278.469} C_VEL
LIN {X 0,Y 575.129,Z 444.169,A -85,B 0,C 180,E1 -2279.818,E2 -2279.818} C_VEL
LIN {X 0,Y 573.3,Z 436.52,A -85,B 0,C 180,E1 -2280.988,E2 -2280.988} C_VEL
LIN {X 0,Y 573.258,Z 436.319,A -85,B 0,C 180,E1 -2283.523,E2 -2283.523} C_VEL
LIN {X 0,Y 573.257,Z 436.326,A -85,B 0,C 180,E1 -2286.047,E2 -2286.047} C_VEL
LIN {X 0,Y 573.243,Z 436.318,A -85,B 0,C 180,E1 -2288.7,E2 -2288.7} C_VEL
LIN {X 0,Y 573.229,Z 436.333,A -85,B 0,C 180,E1 -2291.456,E2 -2291.456} C_VEL
LIN {X 0,Y 573.229,Z 436.327,A -85,B 0,C 180,E1 -2294.333,E2 -2294.333} C_VEL
LIN {X 0,Y 573.238,Z 436.327,A -85,B 0,C 180,E1 -2297.357,E2 -2297.357} C_VEL
LIN {X 0,Y 573.243,Z 436.324,A -85,B 0,C 180,E1 -2300.393,E2 -2300.393} C_VEL
LIN {X 0,Y 573.25,Z 436.323,A -85,B 0,C 180,E1 -2303.077,E2 -2303.077} C_VEL
LIN {X 0,Y 573.266,Z 436.322,A -85,B 0,C 180,E1 -2305.671,E2 -2305.671} C_VEL
LIN {X 0,Y 573.241,Z 436.33,A -85,B 0,C 180,E1 -2308.185,E2 -2308.185} C_VEL
LIN {X 0,Y 573.26,Z 436.317,A -85,B 0,C 180,E1 -2310.634,E2 -2310.634} C_VEL
LIN {X 0,Y 573.261,Z 436.32,A -85,B 0,C 180,E1 -2313.5,E2 -2313.5} C_VEL
LIN {X 0,Y 573.225,Z 436.335,A -85,B 0,C 180,E1 -2316.134,E2 -2316.134} C_VEL
LIN {X 0,Y 573.252,Z 436.315,A -85,B 0,C 180,E1 -2319.174,E2 -2319.174} C_VEL
LIN {X 0,Y 573.23,Z 436.32,A -85,B 0,C 180,E1 -2321.411,E2 -2321.411} C_VEL
LIN {X 0,Y 573.249,Z 436.323,A -85,B 0,C 180,E1 -2323.622,E2 -2323.622} C_VEL
LIN {X 0,Y 573.227,Z 436.329,A -85,B 0,C 180,E1 -2326.529,E2 -2326.529} C_VEL
LIN {X 0,Y 573.274,Z 436.323,A -85,B 0,C 180,E1 -2328.734,E2 -2328.734} C_VEL
LIN {X 0,Y 573.299,Z 436.314,A -85,B 0,C 180,E1 -2331.541,E2 -2331.541} C_VEL
LIN {X 0,Y 573.282,Z 436.329,A -85,B 0,C 180,E1 -2334.372,E2 -2334.372} C_VEL
LIN {X 0,Y 573.3,Z 436.317,A -85,B 0,C 180,E1 -2337.892,E2 -2337.892} C_VEL
LIN {X 0,Y 573.328,Z 436.317,A -85,B 0,C 180,E1 -2340.702,E2 -2340.702} C_VEL
LIN {X 0,Y 573.231,Z 436.324,A -85,B 0,C 180,E1 -2343.514,E2 -2343.514} C_VEL
LIN {X 0,Y 573.289,Z 436.316,A -85,B 0,C 180,E1 -2345.628,E2 -2345.628} C_VEL
LIN {X 0,Y 573.299,Z 436.323,A -85,B 0,C 180,E1 -2348.459,E2 -2348.459} C_VEL
LIN {X 0,Y 573.289,Z 436.317,A -85,B 0,C 180,E1 -2351.311,E2 -2351.311} C_VEL
LIN {X 0,Y 573.27,Z 436.325,A -85,B 0,C 180,E1 -2354.425,E2 -2354.425} C_VEL
LIN {X 0,Y 573.249,Z 436.327,A -85,B 0,C 180,E1 -2357.112,E2 -2357.112} C_VEL
LIN {X 0,Y 573.247,Z 436.322,A -85,B 0,C 180,E1 -2360.077,E2 -2360.077} C_VEL
LIN {X 0,Y 573.228,Z 436.328,A -85,B 0,C 180,E1 -2362.338,E2 -2362.338} C_VEL
LIN {X 0,Y 573.242,Z 436.325,A -85,B 0,C 180,E1 -2364.399,E2 -2364.399} C_VEL
LIN {X 0,Y 572.616,Z 436.409,A -85,B 0,C 180,E1 -2364.986,E2 -2364.986} C_VEL
LIN {X 0,Y 569.778,Z 436.764,A -85,B 0,C 180,E1 -2365.937,E2 -2365.937} C_VEL
LIN {X 0,Y 567.35,Z 437.062,A -85,B 0,C 180,E1 -2366.703,E2 -2366.703} C_VEL
LIN {X 0,Y 566.298,Z 437.189,A -85,B 0,C 180,E1 -2367.295,E2 -2367.295} C_VEL
LIN {X 0,Y 566.208,Z 437.198,A -85,B 0,C 180,E1 -2367.495,E2 -2367.495} C_VEL
LIN {X 0,Y 566.185,Z 437.207,A -85,B 0,C 180,E1 -2370.592,E2 -2370.592} C_VEL
LIN {X 0,Y 566.219,Z 437.199,A -85,B 0,C 180,E1 -2373.102,E2 -2373.102} C_VEL
LIN {X 0,Y 566.203,Z 437.201,A -85,B 0,C 180,E1 -2375.689,E2 -2375.689} C_VEL
LIN {X 0,Y 566.21,Z 437.202,A -85,B 0,C 180,E1 -2378.56,E2 -2378.56} C_VEL
LIN {X 0,Y 566.212,Z 437.209,A -85,B 0,C 180,E1 -2381.136,E2 -2381.136} C_VEL
LIN {X 0,Y 566.192,Z 437.203,A -85,B 0,C 180,E1 -2384.036,E2 -2384.036} C_VEL
LIN {X 0,Y 566.197,Z 437.209,A -85,B 0,C 180,E1 -2387.083,E2 -2387.083} C_VEL
LIN {X 0,Y 566.219,Z 437.202,A -85,B 0,C 180,E1 -2389.803,E2 -2389.803} C_VEL
LIN {X 0,Y 566.192,Z 437.203,A -85,B 0,C 180,E1 -2392.599,E2 -2392.599} C_VEL
LIN {X 0,Y 566.215,Z 437.205,A -85,B 0,C 180,E1 -2395.184,E2 -2395.184} C_VEL
LIN {X 0,Y 566.23,Z 437.203,A -85,B 0,C 180,E1 -2397.744,E2 -2397.744} C_VEL
LIN {X 0,Y 566.198,Z 437.202,A -85,B 0,C 180,E1 -2400.328,E2 -2400.328} C_VEL
LIN {X 0,Y 566.22,Z 437.199,A -85,B 0,C 180,E1 -2402.662,E2 -2402.662} C_VEL
LIN {X 0,Y 566.231,Z 437.2,A -85,B 0,C 180,E1 -2405.039,E2 -2405.039} C_VEL
LIN {X 0,Y 566.19,Z 437.205,A -85,B 0,C 180,E1 -2408.138,E2 -2408.138} C_VEL
LIN {X 0,Y 566.232,Z 437.198,A -85,B 0,C 180,E1 -2410.612,E2 -2410.612} C_VEL
LIN {X 0,Y 566.216,Z 437.204,A -85,B 0,C 180,E1 -2413.413,E2 -2413.413} C_VEL
LIN {X 0,Y 566.197,Z 437.204,A -85,B 0,C 180,E1 -2416.359,E2 -2416.359} C_VEL
LIN {X 0,Y 566.231,Z 437.198,A -85,B 0,C 180,E1 -2418.675,E2 -2418.675} C_VEL
LIN {X 0,Y 566.225,Z 437.202,A -85,B 0,C 180,E1 -2421.434,E2 -2421.434} C_VEL
LIN {X 0,Y 566.255,Z 437.199,A -85,B 0,C 180,E1 -2424.302,E2 -2424.302} C_VEL
LIN {X 0,Y 566.28,Z 437.201,A -85,B 0,C 180,E1 -2427.866,E2 -2427.866} C_VEL
LIN {X 0,Y 566.297,Z 437.191,A -85,B 0,C 180,E1 -2430.711,E2 -2430.711} C_VEL
LIN {X 0,Y 566.268,Z 437.194,A -85,B 0,C 180,E1 -2432.846,E2 -2432.846} C_VEL
LIN {X 0,Y 566.255,Z 437.199,A -85,B 0,C 180,E1 -2435.698,E2 -2435.698} C_VEL
LIN {X 0,Y 566.225,Z 437.202,A -85,B 0,C 180,E1 -2438.566,E2 -2438.566} C_VEL
LIN {X 0,Y 566.238,Z 437.198,A -85,B 0,C 180,E1 -2441.454,E2 -2441.454} C_VEL
LIN {X 0,Y 566.231,Z 437.204,A -85,B 0,C 180,E1 -2444.507,E2 -2444.507} C_VEL
LIN {X 0,Y 566.2,Z 437.201,A -85,B 0,C 180,E1 -2447.331,E2 -2447.331} C_VEL
LIN {X 0,Y 566.21,Z 437.209,A -85,B 0,C 180,E1 -2450.337,E2 -2450.337} C_VEL
LIN {X 0,Y 566.168,Z 437.206,A -85,B 0,C 180,E1 -2453.282,E2 -2453.282} C_VEL
LIN {X 0,Y 566.22,Z 437.2,A -85,B 0,C 180,E1 -2455.748,E2 -2455.748} C_VEL
LIN {X 0,Y 566.202,Z 437.207,A -85,B 0,C 180,E1 -2458.203,E2 -2458.203} C_VEL
LIN {X 0,Y 566.192,Z 437.204,A -85,B 0,C 180,E1 -2461.077,E2 -2461.077} C_VEL
LIN {X 0,Y 566.223,Z 437.199,A -85,B 0,C 180,E1 -2463.737,E2 -2463.737} C_VEL
LIN {X 0,Y 566.21,Z 437.21,A -85,B 0,C 180,E1 -2466.568,E2 -2466.568} C_VEL
LIN {X 0,Y 566.205,Z 437.2,A -85,B 0,C 180,E1 -2469.685,E2 -2469.685} C_VEL
LIN {X 0,Y 566.206,Z 437.202,A -85,B 0,C 180,E1 -2472.087,E2 -2472.087} C_VEL
LIN {X 0,Y 566.166,Z 437.211,A -85,B 0,C 180,E1 -2475.035,E2 -2475.035} C_VEL
LIN {X 0,Y 566.216,Z 437.2,A -85,B 0,C 180,E1 -2478.135,E2 -2478.135} C_VEL
LIN {X 0,Y 566.215,Z 437.208,A -85,B 0,C 180,E1 -2480.727,E2 -2480.727} C_VEL
LIN {X 0,Y 566.209,Z 437.199,A -85,B 0,C 180,E1 -2483.783,E2 -2483.783} C_VEL
LIN {X 0,Y 566.202,Z 437.193,A -85,B 0,C 180,E1 -2486.265,E2 -2486.265} C_VEL
LIN {X 0,Y 566.194,Z 437.21,A -85,B 0,C 180,E1 -2488.921,E2 -2488.921} C_VEL
LIN {X 0,Y 566.187,Z 437.209,A -85,B 0,C 180,E1 -2491.047,E2 -2491.047} C_VEL
LIN {X 0,Y 566.237,Z 437.193,A -85,B 0,C 180,E1 -2493.46,E2 -2493.46} C_VEL
LIN {X 0,Y 566.19,Z 437.202,A -85,B 0,C 180,E1 -2495.819,E2 -2495.819} C_VEL
LIN {X 0,Y 566.207,Z 437.206,A -85,B 0,C 180,E1 -2498.903,E2 -2498.903} C_VEL
LIN {X 0,Y 566.204,Z 437.209,A -85,B 0,C 180,E1 -2501.173,E2 -2501.173} C_VEL
LIN {X 0,Y 566.21,Z 437.204,A -85,B 0,C 180,E1 -2503.412,E2 -2503.412} C_VEL
LIN {X 0,Y 566.19,Z 437.202,A -85,B 0,C 180,E1 -2506.359,E2 -2506.359} C_VEL
LIN {X 0,Y 566.265,Z 437.191,A -85,B 0,C 180,E1 -2508.654,E2 -2508.654} C_VEL
LIN {X 0,Y 566.24,Z 437.204,A -85,B 0,C 180,E1 -2511.435,E2 -2511.435} C_VEL
LIN {X 0,Y 566.258,Z 437.192,A -85,B 0,C 180,E1 -2514.302,E2 -2514.302} C_VEL
LIN {X 0,Y 566.271,Z 437.193,A -85,B 0,C 180,E1 -2517.866,E2 -2517.866} C_VEL
LIN {X 0,Y 566.298,Z 437.189,A -85,B 0,C 180,E1 -2520.711,E2 -2520.711} C_VEL
LIN {X 0,Y 566.271,Z 437.192,A -85,B 0,C 180,E1 -2522.846,E2 -2522.846} C_VEL
LIN {X 0,Y 566.25,Z 437.203,A -85,B 0,C 180,E1 -2525.698,E2 -2525.698} C_VEL
LIN {X 0,Y 566.24,Z 437.192,A -85,B 0,C 180,E1 -2528.566,E2 -2528.566} C_VEL
LIN {X 0,Y 566.241,Z 437.201,A -85,B 0,C 180,E1 -2531.454,E2 -2531.454} C_VEL
LIN {X 0,Y 566.224,Z 437.198,A -85,B 0,C 180,E1 -2534.507,E2 -2534.507} C_VEL
LIN {X 0,Y 566.195,Z 437.203,A -85,B 0,C 180,E1 -2537.332,E2 -2537.332} C_VEL
LIN {X 0,Y 566.21,Z 437.194,A -85,B 0,C 180,E1 -2540.337,E2 -2540.337} C_VEL
LIN {X 0,Y 566.181,Z 437.205,A -85,B 0,C 180,E1 -2543.404,E2 -2543.404} C_VEL
LIN {X 0,Y 566.216,Z 437.206,A -85,B 0,C 180,E1 -2545.749,E2 -2545.749} C_VEL
LIN {X 0,Y 566.197,Z 437.2,A -85,B 0,C 180,E1 -2548.203,E2 -2548.203} C_VEL
LIN {X 0,Y 566.186,Z 437.204,A -85,B 0,C 180,E1 -2550.592,E2 -2550.592} C_VEL
LIN {X 0,Y 566.221,Z 437.198,A -85,B 0,C 180,E1 -2553.102,E2 -2553.102} C_VEL
LIN {X 0,Y 566.204,Z 437.199,A -85,B 0,C 180,E1 -2555.689,E2 -2555.689} C_VEL
LIN {X 0,Y 566.211,Z 437.202,A -85,B 0,C 180,E1 -2558.56,E2 -2558.56} C_VEL
LIN {X 0,Y 566.206,Z 437.2,A -85,B 0,C 180,E1 -2561.137,E2 -2561.137} C_VEL
LIN {X 0,Y 566.194,Z 437.208,A -85,B 0,C 180,E1 -2564.036,E2 -2564.036} C_VEL
LIN {X 0,Y 566.195,Z 437.201,A -85,B 0,C 180,E1 -2567.083,E2 -2567.083} C_VEL
LIN {X 0,Y 566.222,Z 437.202,A -85,B 0,C 180,E1 -2569.803,E2 -2569.803} C_VEL
LIN {X 0,Y 566.194,Z 437.2,A -85,B 0,C 180,E1 -2572.6,E2 -2572.6} C_VEL
LIN {X 0,Y 566.216,Z 437.197,A -85,B 0,C 180,E1 -2575.184,E2 -2575.184} C_VEL
LIN {X 0,Y 566.232,Z 437.204,A -85,B 0,C 180,E1 -2577.744,E2 -2577.744} C_VEL
LIN {X 0,Y 566.234,Z 437.348,A -85,B 0,C 180,E1 -2578.682,E2 -2578.682} C_VEL
LIN {X 0,Y 568.463,Z 446.592,A -85,B 0,C 180,E1 -2580.127,E2 -2580.127} C_VEL
LIN {X 0,Y 567.946,Z 470.109,A -85,B 0,C 180,E1 -2583.263,E2 -2583.263} C_VEL
LIN {X 0,Y 567.735,Z 484.208,A -85,B 0,C 180,E1 -2585.082,E2 -2585.082} C_VEL
LIN {X 0,Y 569.675,Z 492.164,A -85,B 0,C 180,E1 -2585.309,E2 -2585.309} C_VEL
LIN {X 0,Y 569.974,Z 496.031,A -85,B 0,C 180,E1 -2585.375,E2 -2585.375} C_VEL
LIN {X 0,Y 569.138,Z 695.098,A -85,B 0,C 180,E1 -2588.034,E2 -2588.034} C_VEL
LIN {X 0,Y 568.921,Z 711.367,A -85,B 0,C 180,E1 -2588.367,E2 -2588.367} C_VEL
LIN {X 0,Y 568.664,Z 729.313,A -85,B 0,C 180,E1 -2588.903,E2 -2588.903} C_VEL
LIN {X 0,Y 568.394,Z 744.679,A -85,B 0,C 180,E1 -2589.509,E2 -2589.509} C_VEL
LIN {X 0,Y 568.096,Z 758.846,A -85,B 0,C 180,E1 -2590.199,E2 -2590.199} C_VEL
LIN {X 0,Y 567.748,Z 773.335,A -85,B 0,C 180,E1 -2591.038,E2 -2591.038} C_VEL
LIN {X 0,Y 567.408,Z 788.133,A -85,B 0,C 180,E1 -2592.065,E2 -2592.065} C_VEL
LIN {X 0,Y 567.052,Z 802.46,A -85,B 0,C 180,E1 -2593.253,E2 -2593.253} C_VEL
LIN {X 0,Y 566.804,Z 813.828,A -85,B 0,C 180,E1 -2594.355,E2 -2594.355} C_VEL
LIN {X 0,Y 566.558,Z 825.314,A -85,B 0,C 180,E1 -2595.636,E2 -2595.636} C_VEL
LIN {X 0,Y 566.337,Z 836.438,A -85,B 0,C 180,E1 -2597.093,E2 -2597.093} C_VEL
LIN {X 0,Y 566.207,Z 845.813,A -85,B 0,C 180,E1 -2598.545,E2 -2598.545} C_VEL
LIN {X 0,Y 566.083,Z 853.665,A -85,B 0,C 180,E1 -2599.991,E2 -2599.991} C_VEL
LIN {X 0,Y 565.998,Z 860.285,A -85,B 0,C 180,E1 -2601.431,E2 -2601.431} C_VEL
LIN {X 0,Y 565.965,Z 865.667,A -85,B 0,C 180,E1 -2602.867,E2 -2602.867} C_VEL
LIN {X 0,Y 565.962,Z 870.027,A -85,B 0,C 180,E1 -2604.299,E2 -2604.299} C_VEL
LIN {X 0,Y 565.908,Z 873.297,A -85,B 0,C 180,E1 -2605.727,E2 -2605.727} C_VEL
LIN {X 0,Y 565.868,Z 875.656,A -85,B 0,C 180,E1 -2607.152,E2 -2607.152} C_VEL
LIN {X 0,Y 565.838,Z 877.006,A -85,B 0,C 180,E1 -2608.577,E2 -2608.577} C_VEL
LIN {X 0,Y 565.834,Z 877.5,A -85,B 0,C 180,E1 -2610,E2 -2610} C_VEL
LIN {X 0,Y 565.838,Z 877.006,A -85,B 0,C 180,E1 -2611.423,E2 -2611.423} C_VEL
LIN {X 0,Y 565.868,Z 875.656,A -85,B 0,C 180,E1 -2612.848,E2 -2612.848} C_VEL
LIN {X 0,Y 565.908,Z 873.297,A -85,B 0,C 180,E1 -2614.273,E2 -2614.273} C_VEL
LIN {X 0,Y 565.962,Z 870.027,A -85,B 0,C 180,E1 -2615.701,E2 -2615.701} C_VEL
LIN {X 0,Y 565.969,Z 864.423,A -85,B 0,C 180,E1 -2617.492,E2 -2617.492} C_VEL
LIN {X 0,Y 565.994,Z 858.757,A -85,B 0,C 180,E1 -2618.929,E2 -2618.929} C_VEL
LIN {X 0,Y 566.092,Z 851.847,A -85,B 0,C 180,E1 -2620.37,E2 -2620.37} C_VEL
LIN {X 0,Y 566.237,Z 842.48,A -85,B 0,C 180,E1 -2621.999,E2 -2621.999} C_VEL
LIN {X 0,Y 566.401,Z 832.44,A -85,B 0,C 180,E1 -2623.453,E2 -2623.453} C_VEL
LIN {X 0,Y 566.636,Z 821.881,A -85,B 0,C 180,E1 -2624.77,E2 -2624.77} C_VEL
LIN {X 0,Y 566.868,Z 810.274,A -85,B 0,C 180,E1 -2626.013,E2 -2626.013} C_VEL
